LIN {X 0,Y 554.987,Z 579.027,A -85,B 0,C 180,E1 25629.323,E2 25629.323} C_VEL
LIN {X 0,Y 555.409,Z 560.565,A -85,B 0,C 180,E1 25628.677,E2 25628.677} C_VEL
LIN {X 0,Y 555.693,Z 541.746,A -85,B 0,C 180,E1 25628.23,E2 25628.23} C_VEL
LIN {X 0,Y 556.819,Z 343.095,A -85,B 0,C 180,E1 25625.485,E2 25625.485} C_VEL
LIN {X 0,Y 555.247,Z 334.788,A -85,B 0,C 180,E1 25625.25,E2 25625.25} C_VEL
LIN {X 0,Y 556.018,Z 305.385,A -85,B 0,C 180,E1 25622.475,E2 25622.475} C_VEL
LIN {X 0,Y 552.345,Z 293.887,A -85,B 0,C 180,E1 25621.069,E2 25621.069} C_VEL
LIN {X 0,Y 552.34,Z 293.681,A -85,B 0,C 180,E1 25617.846,E2 25617.846} C_VEL
LIN {X 0,Y 552.335,Z 293.677,A -85,B 0,C 180,E1 25614.474,E2 25614.474} C_VEL
LIN {X 0,Y 552.308,Z 293.678,A -85,B 0,C 180,E1 25611.119,E2 25611.119} C_VEL
LIN {X 0,Y 552.34,Z 293.682,A -85,B 0,C 180,E1 25607.811,E2 25607.811} C_VEL
LIN {X 0,Y 552.322,Z 293.677,A -85,B 0,C 180,E1 25604.474,E2 25604.474} C_VEL
LIN {X 0,Y 552.301,Z 293.684,A -85,B 0,C 180,E1 25601.084,E2 25601.084} C_VEL
LIN {X 0,Y 552.345,Z 293.682,A -85,B 0,C 180,E1 25597.855,E2 25597.855} C_VEL
LIN {X 0,Y 552.302,Z 293.681,A -85,B 0,C 180,E1 25594.545,E2 25594.545} C_VEL
LIN {X 0,Y 552.297,Z 293.685,A -85,B 0,C 180,E1 25591.099,E2 25591.099} C_VEL
LIN {X 0,Y 552.344,Z 293.681,A -85,B 0,C 180,E1 25587.842,E2 25587.842} C_VEL
LIN {X 0,Y 552.285,Z 293.679,A -85,B 0,C 180,E1 25584.607,E2 25584.607} C_VEL
LIN {X 0,Y 552.314,Z 293.685,A -85,B 0,C 180,E1 25581.338,E2 25581.338} C_VEL
LIN {X 0,Y 552.292,Z 293.682,A -85,B 0,C 180,E1 25578.252,E2 25578.252} C_VEL
LIN {X 0,Y 552.278,Z 293.681,A -85,B 0,C 180,E1 25574.897,E2 25574.897} C_VEL
LIN {X 0,Y 552.337,Z 293.685,A -85,B 0,C 180,E1 25571.676,E2 25571.676} C_VEL
LIN {X 0,Y 552.267,Z 293.68,A -85,B 0,C 180,E1 25568.433,E2 25568.433} C_VEL
LIN {X 0,Y 552.298,Z 293.687,A -85,B 0,C 180,E1 25565.194,E2 25565.194} C_VEL
LIN {X 0,Y 552.276,Z 293.682,A -85,B 0,C 180,E1 25562.075,E2 25562.075} C_VEL
LIN {X 0,Y 552.263,Z 293.686,A -85,B 0,C 180,E1 25558.755,E2 25558.755} C_VEL
LIN {X 0,Y 552.326,Z 293.685,A -85,B 0,C 180,E1 25555.536,E2 25555.536} C_VEL
LIN {X 0,Y 552.265,Z 293.683,A -85,B 0,C 180,E1 25552.406,E2 25552.406} C_VEL
LIN {X 0,Y 552.318,Z 293.686,A -85,B 0,C 180,E1 25549.148,E2 25549.148} C_VEL
LIN {X 0,Y 552.281,Z 293.681,A -85,B 0,C 180,E1 25546.014,E2 25546.014} C_VEL
LIN {X 0,Y 552.279,Z 293.683,A -85,B 0,C 180,E1 25542.566,E2 25542.566} C_VEL
LIN {X 0,Y 552.342,Z 293.686,A -85,B 0,C 180,E1 25539.33,E2 25539.33} C_VEL
LIN {X 0,Y 552.285,Z 293.683,A -85,B 0,C 180,E1 25536.096,E2 25536.096} C_VEL
LIN {X 0,Y 552.309,Z 293.68,A -85,B 0,C 180,E1 25532.741,E2 25532.741} C_VEL
LIN {X 0,Y 552.327,Z 293.686,A -85,B 0,C 180,E1 25529.504,E2 25529.504} C_VEL
LIN {X 0,Y 552.292,Z 293.684,A -85,B 0,C 180,E1 25526.195,E2 25526.195} C_VEL
LIN {X 0,Y 552.345,Z 293.677,A -85,B 0,C 180,E1 25522.93,E2 25522.93} C_VEL
LIN {X 0,Y 552.318,Z 293.684,A -85,B 0,C 180,E1 25519.603,E2 25519.603} C_VEL
LIN {X 0,Y 552.305,Z 293.684,A -85,B 0,C 180,E1 25516.245,E2 25516.245} C_VEL
LIN {X 0,Y 552.341,Z 293.676,A -85,B 0,C 180,E1 25513.002,E2 25513.002} C_VEL
LIN {X 0,Y 552.312,Z 293.674,A -85,B 0,C 180,E1 25509.702,E2 25509.702} C_VEL
LIN {X 0,Y 552.379,Z 293.923,A -85,B 0,C 180,E1 25506.704,E2 25506.704} C_VEL
LIN {X 0,Y 554.146,Z 298.811,A -85,B 0,C 180,E1 25506.242,E2 25506.242} C_VEL
LIN {X 0,Y 559.158,Z 310.667,A -85,B 0,C 180,E1 25505.196,E2 25505.196} C_VEL
LIN {X 0,Y 558.362,Z 353.988,A -85,B 0,C 180,E1 25502.614,E2 25502.614} C_VEL
LIN {X 0,Y 557.656,Z 390.963,A -85,B 0,C 180,E1 25500.436,E2 25500.436} C_VEL
LIN {X 0,Y 558.742,Z 400.337,A -85,B 0,C 180,E1 25500.232,E2 25500.232} C_VEL
LIN {X 0,Y 557.381,Z 635.152,A -85,B 0,C 180,E1 25496.937,E2 25496.937} C_VEL
LIN {X 0,Y 557.116,Z 659.61,A -85,B 0,C 180,E1 25496.529,E2 25496.529} C_VEL
LIN {X 0,Y 556.72,Z 680.633,A -85,B 0,C 180,E1 25495.975,E2 25495.975} C_VEL
LIN {X 0,Y 556.289,Z 700.028,A -85,B 0,C 180,E1 25495.274,E2 25495.274} C_VEL
LIN {X 0,Y 555.753,Z 719.239,A -85,B 0,C 180,E1 25494.386,E2 25494.386} C_VEL
LIN {X 0,Y 555.148,Z 738.316,A -85,B 0,C 180,E1 25493.286,E2 25493.286} C_VEL
LIN {X 0,Y 554.551,Z 756.388,A -85,B 0,C 180,E1 25492.025,E2 25492.025} C_VEL
LIN {X 0,Y 553.976,Z 773.443,A -85,B 0,C 180,E1 25490.606,E2 25490.606} C_VEL
LIN {X 0,Y 553.441,Z 789.448,A -85,B 0,C 180,E1 25489.031,E2 25489.031} C_VEL
LIN {X 0,Y 552.984,Z 804.238,A -85,B 0,C 180,E1 25487.315,E2 25487.315} C_VEL
LIN {X 0,Y 552.622,Z 817.278,A -85,B 0,C 180,E1 25485.531,E2 25485.531} C_VEL
LIN {X 0,Y 552.359,Z 828.534,A -85,B 0,C 180,E1 25483.717,E2 25483.717} C_VEL
LIN {X 0,Y 552.147,Z 838.91,A -85,B 0,C 180,E1 25481.701,E2 25481.701} C_VEL
LIN {X 0,Y 552.024,Z 847.28,A -85,B 0,C 180,E1 25479.697,E2 25479.697} C_VEL
LIN {X 0,Y 551.959,Z 854.202,A -85,B 0,C 180,E1 25477.599,E2 25477.599} C_VEL
LIN {X 0,Y 551.92,Z 859.556,A -85,B 0,C 180,E1 25475.405,E2 25475.405} C_VEL
LIN {X 0,Y 551.909,Z 862.942,A -85,B 0,C 180,E1 25473.323,E2 25473.323} C_VEL
LIN {X 0,Y 551.911,Z 864.759,A -85,B 0,C 180,E1 25471.142,E2 25471.142} C_VEL
LIN {X 0,Y 551.915,Z 864.783,A -85,B 0,C 180,E1 25468.962,E2 25468.962} C_VEL
LIN {X 0,Y 551.914,Z 863.169,A -85,B 0,C 180,E1 25466.885,E2 25466.885} C_VEL
LIN {X 0,Y 551.921,Z 859.76,A -85,B 0,C 180,E1 25464.699,E2 25464.699} C_VEL
LIN {X 0,Y 551.952,Z 854.809,A -85,B 0,C 180,E1 25462.611,E2 25462.611} C_VEL
LIN {X 0,Y 552.022,Z 848.49,A -85,B 0,C 180,E1 25460.618,E2 25460.618} C_VEL
LIN {X 0,Y 552.138,Z 839.875,A -85,B 0,C 180,E1 25458.51,E2 25458.51} C_VEL
LIN {X 0,Y 552.321,Z 830.266,A -85,B 0,C 180,E1 25456.602,E2 25456.602} C_VEL
LIN {X 0,Y 552.585,Z 818.607,A -85,B 0,C 180,E1 25454.67,E2 25454.67} C_VEL
LIN {X 0,Y 552.945,Z 805.602,A -85,B 0,C 180,E1 25452.858,E2 25452.858} C_VEL
LIN {X 0,Y 553.393,Z 790.965,A -85,B 0,C 180,E1 25451.131,E2 25451.131} C_VEL
LIN {X 0,Y 553.892,Z 775.855,A -85,B 0,C 180,E1 25449.611,E2 25449.611} C_VEL
LIN {X 0,Y 554.455,Z 759.284,A -85,B 0,C 180,E1 25448.193,E2 25448.193} C_VEL
LIN {X 0,Y 555.07,Z 740.902,A -85,B 0,C 180,E1 25446.879,E2 25446.879} C_VEL
LIN {X 0,Y 555.652,Z 722.284,A -85,B 0,C 180,E1 25445.779,E2 25445.779} C_VEL
LIN {X 0,Y 556.159,Z 704.004,A -85,B 0,C 180,E1 25444.896,E2 25444.896} C_VEL
LIN {X 0,Y 556.654,Z 683.569,A -85,B 0,C 180,E1 25444.118,E2 25444.118} C_VEL
LIN {X 0,Y 557.081,Z 663.506,A -85,B 0,C 180,E1 25443.556,E2 25443.556} C_VEL
LIN {X 0,Y 557.344,Z 642.37,A -85,B 0,C 180,E1 25443.163,E2 25443.163} C_VEL
LIN {X 0,Y 558.712,Z 404.697,A -85,B 0,C 180,E1 25439.829,E2 25439.829} C_VEL
LIN {X 0,Y 558.481,Z 396.637,A -85,B 0,C 180,E1 25439.698,E2 25439.698} C_VEL
LIN {X 0,Y 557.585,Z 389.593,A -85,B 0,C 180,E1 25439.505,E2 25439.505} C_VEL
LIN {X 0,Y 558.839,Z 332.018,A -85,B 0,C 180,E1 25436.068,E2 25436.068} C_VEL
LIN {X 0,Y 558.964,Z 309.864,A -85,B 0,C 180,E1 25434.743,E2 25434.743} C_VEL
LIN {X 0,Y 552.405,Z 294.092,A -85,B 0,C 180,E1 25433.324,E2 25433.324} C_VEL
LIN {X 0,Y 552.339,Z 293.671,A -85,B 0,C 180,E1 25432.969,E2 25432.969} C_VEL
LIN {X 0,Y 552.316,Z 293.676,A -85,B 0,C 180,E1 25429.653,E2 25429.653} C_VEL
LIN {X 0,Y 552.31,Z 293.676,A -85,B 0,C 180,E1 25426.246,E2 25426.246} C_VEL
LIN {X 0,Y 552.344,Z 293.682,A -85,B 0,C 180,E1 25423.004,E2 25423.004} C_VEL
LIN {X 0,Y 552.302,Z 293.683,A -85,B 0,C 180,E1 25419.702,E2 25419.702} C_VEL
LIN {X 0,Y 552.307,Z 293.672,A -85,B 0,C 180,E1 25416.297,E2 25416.297} C_VEL
LIN {X 0,Y 552.34,Z 293.682,A -85,B 0,C 180,E1 25413.016,E2 25413.016} C_VEL
LIN {X 0,Y 552.29,Z 293.685,A -85,B 0,C 180,E1 25409.739,E2 25409.739} C_VEL
LIN {X 0,Y 552.326,Z 293.687,A -85,B 0,C 180,E1 25406.444,E2 25406.444} C_VEL
LIN {X 0,Y 552.304,Z 293.681,A -85,B 0,C 180,E1 25403.244,E2 25403.244} C_VEL
LIN {X 0,Y 552.284,Z 293.685,A -85,B 0,C 180,E1 25399.898,E2 25399.898} C_VEL
LIN {X 0,Y 552.345,Z 293.684,A -85,B 0,C 180,E1 25396.619,E2 25396.619} C_VEL
LIN {X 0,Y 552.277,Z 293.679,A -85,B 0,C 180,E1 25393.399,E2 25393.399} C_VEL
LIN {X 0,Y 552.284,Z 293.685,A -85,B 0,C 180,E1 25389.992,E2 25389.992} C_VEL
LIN {X 0,Y 552.307,Z 293.682,A -85,B 0,C 180,E1 25386.862,E2 25386.862} C_VEL
LIN {X 0,Y 552.263,Z 293.684,A -85,B 0,C 180,E1 25383.633,E2 25383.633} C_VEL
LIN {X 0,Y 552.332,Z 293.688,A -85,B 0,C 180,E1 25380.415,E2 25380.415} C_VEL
LIN {X 0,Y 552.261,Z 293.683,A -85,B 0,C 180,E1 25377.198,E2 25377.198} C_VEL
LIN {X 0,Y 552.27,Z 293.687,A -85,B 0,C 180,E1 25373.764,E2 25373.764} C_VEL
LIN {X 0,Y 552.286,Z 293.681,A -85,B 0,C 180,E1 25370.833,E2 25370.833} C_VEL
LIN {X 0,Y 552.268,Z 293.686,A -85,B 0,C 180,E1 25367.558,E2 25367.558} C_VEL
LIN {X 0,Y 552.34,Z 293.683,A -85,B 0,C 180,E1 25364.352,E2 25364.352} C_VEL
LIN {X 0,Y 552.276,Z 293.684,A -85,B 0,C 180,E1 25361.091,E2 25361.091} C_VEL
LIN {X 0,Y 552.301,Z 293.685,A -85,B 0,C 180,E1 25357.767,E2 25357.767} C_VEL
LIN {X 0,Y 552.312,Z 293.681,A -85,B 0,C 180,E1 25354.593,E2 25354.593} C_VEL
LIN {X 0,Y 552.299,Z 293.687,A -85,B 0,C 180,E1 25352.738,E2 25352.738} C_VEL
LIN {X 0,Y 551.36,Z 293.809,A -85,B 0,C 180,E1 25351.938,E2 25351.938} C_VEL
LIN {X 0,Y 544.881,Z 294.609,A -85,B 0,C 180,E1 25349.694,E2 25349.694} C_VEL
LIN {X 0,Y 544.346,Z 294.673,A -85,B 0,C 180,E1 25349.109,E2 25349.109} C_VEL
LIN {X 0,Y 544.389,Z 294.67,A -85,B 0,C 180,E1 25345.804,E2 25345.804} C_VEL
LIN {X 0,Y 544.381,Z 294.675,A -85,B 0,C 180,E1 25342.507,E2 25342.507} C_VEL
LIN {X 0,Y 544.357,Z 294.672,A -85,B 0,C 180,E1 25339.164,E2 25339.164} C_VEL
LIN {X 0,Y 544.405,Z 294.667,A -85,B 0,C 180,E1 25335.887,E2 25335.887} C_VEL
LIN {X 0,Y 544.376,Z 294.665,A -85,B 0,C 180,E1 25332.523,E2 25332.523} C_VEL
LIN {X 0,Y 544.368,Z 294.665,A -85,B 0,C 180,E1 25329.184,E2 25329.184} C_VEL
LIN {X 0,Y 544.404,Z 294.669,A -85,B 0,C 180,E1 25325.864,E2 25325.864} C_VEL
LIN {X 0,Y 544.38,Z 294.676,A -85,B 0,C 180,E1 25322.537,E2 25322.537} C_VEL
LIN {X 0,Y 544.416,Z 294.861,A -85,B 0,C 180,E1 25319.297,E2 25319.297} C_VEL
LIN {X 0,Y 548.778,Z 308.855,A -85,B 0,C 180,E1 25317.566,E2 25317.566} C_VEL
LIN {X 0,Y 548.006,Z 335.919,A -85,B 0,C 180,E1 25315.02,E2 25315.02} C_VEL
LIN {X 0,Y 549.744,Z 345.387,A -85,B 0,C 180,E1 25314.785,E2 25314.785} C_VEL
LIN {X 0,Y 548.559,Z 542.987,A -85,B 0,C 180,E1 25312.041,E2 25312.041} C_VEL
LIN {X 0,Y 548.263,Z 561.882,A -85,B 0,C 180,E1 25311.584,E2 25311.584} C_VEL
LIN {X 0,Y 547.817,Z 579.557,A -85,B 0,C 180,E1 25310.96,E2 25310.96} C_VEL
LIN {X 0,Y 547.296,Z 596.827,A -85,B 0,C 180,E1 25310.146,E2 25310.146} C_VEL
LIN {X 0,Y 546.679,Z 613.249,A -85,B 0,C 180,E1 25309.165,E2 25309.165} C_VEL
LIN {X 0,Y 546.031,Z 629.329,A -85,B 0,C 180,E1 25307.971,E2 25307.971} C_VEL
LIN {X 0,Y 545.411,Z 644.251,A -85,B 0,C 180,E1 25306.617,E2 25306.617} C_VEL
LIN {X 0,Y 544.925,Z 659.491,A -85,B 0,C 180,E1 25304.993,E2 25304.993} C_VEL
LIN {X 0,Y 544.571,Z 672.136,A -85,B 0,C 180,E1 25303.376,E2 25303.376} C_VEL
LIN {X 0,Y 544.302,Z 683.234,A -85,B 0,C 180,E1 25301.657,E2 25301.657} C_VEL
LIN {X 0,Y 544.121,Z 692.806,A -85,B 0,C 180,E1 25299.84,E2 25299.84} C_VEL
LIN {X 0,Y 544.003,Z 700.413,A -85,B 0,C 180,E1 25298.029,E2 25298.029} C_VEL
LIN {X 0,Y 543.946,Z 706.59,A -85,B 0,C 180,E1 25296.12,E2 25296.12} C_VEL
LIN {X 0,Y 543.921,Z 710.996,A -85,B 0,C 180,E1 25294.217,E2 25294.217} C_VEL
LIN {X 0,Y 543.913,Z 713.744,A -85,B 0,C 180,E1 25292.318,E2 25292.318} C_VEL
LIN {X 0,Y 543.909,Z 714.928,A -85,B 0,C 180,E1 25290.316,E2 25290.316} C_VEL
LIN {X 0,Y 543.913,Z 714.376,A -85,B 0,C 180,E1 25288.315,E2 25288.315} C_VEL
LIN {X 0,Y 543.911,Z 712.229,A -85,B 0,C 180,E1 25286.417,E2 25286.417} C_VEL
LIN {X 0,Y 543.932,Z 708.459,A -85,B 0,C 180,E1 25284.515,E2 25284.515} C_VEL
LIN {X 0,Y 543.974,Z 702.972,A -85,B 0,C 180,E1 25282.608,E2 25282.608} C_VEL
LIN {X 0,Y 544.075,Z 695.621,A -85,B 0,C 180,E1 25280.694,E2 25280.694} C_VEL
LIN {X 0,Y 544.235,Z 686.506,A -85,B 0,C 180,E1 25278.831,E2 25278.831} C_VEL
LIN {X 0,Y 544.463,Z 676.445,A -85,B 0,C 180,E1 25277.162,E2 25277.162} C_VEL
LIN {X 0,Y 544.769,Z 664.701,A -85,B 0,C 180,E1 25275.546,E2 25275.546} C_VEL
LIN {X 0,Y 545.161,Z 651.496,A -85,B 0,C 180,E1 25274.032,E2 25274.032} C_VEL
LIN {X 0,Y 545.774,Z 635.715,A -85,B 0,C 180,E1 25272.484,E2 25272.484} C_VEL
LIN {X 0,Y 546.393,Z 620.716,A -85,B 0,C 180,E1 25271.268,E2 25271.268} C_VEL
LIN {X 0,Y 547.021,Z 604.25,A -85,B 0,C 180,E1 25270.181,E2 25270.181} C_VEL
LIN {X 0,Y 547.584,Z 587.755,A -85,B 0,C 180,E1 25269.31,E2 25269.31} C_VEL
LIN {X 0,Y 548.078,Z 569.85,A -85,B 0,C 180,E1 25268.584,E2 25268.584} C_VEL
LIN {X 0,Y 548.441,Z 551.518,A -85,B 0,C 180,E1 25268.051,E2 25268.051} C_VEL
LIN {X 0,Y 548.652,Z 532.068,A -85,B 0,C 180,E1 25267.695,E2 25267.695} C_VEL
LIN {X 0,Y 549.626,Z 343.643,A -85,B 0,C 180,E1 25265.094,E2 25265.094} C_VEL
LIN {X 0,Y 547.949,Z 335.49,A -85,B 0,C 180,E1 25264.869,E2 25264.869} C_VEL
LIN {X 0,Y 548.672,Z 308.058,A -85,B 0,C 180,E1 25262.257,E2 25262.257} C_VEL
LIN {X 0,Y 544.419,Z 294.84,A -85,B 0,C 180,E1 25260.606,E2 25260.606} C_VEL
LIN {X 0,Y 544.375,Z 294.675,A -85,B 0,C 180,E1 25257.193,E2 25257.193} C_VEL
LIN {X 0,Y 544.4,Z 294.672,A -85,B 0,C 180,E1 25253.876,E2 25253.876} C_VEL
LIN {X 0,Y 544.393,Z 294.662,A -85,B 0,C 180,E1 25250.48,E2 25250.48} C_VEL
LIN {X 0,Y 544.367,Z 294.663,A -85,B 0,C 180,E1 25247.127,E2 25247.127} C_VEL
LIN {X 0,Y 544.405,Z 294.671,A -85,B 0,C 180,E1 25243.8,E2 25243.8} C_VEL
LIN {X 0,Y 544.381,Z 294.669,A -85,B 0,C 180,E1 25240.418,E2 25240.418} C_VEL
LIN {X 0,Y 544.36,Z 294.674,A -85,B 0,C 180,E1 25237.046,E2 25237.046} C_VEL
LIN {X 0,Y 544.403,Z 294.67,A -85,B 0,C 180,E1 25233.699,E2 25233.699} C_VEL
LIN {X 0,Y 544.361,Z 294.671,A -85,B 0,C 180,E1 25230.461,E2 25230.461} C_VEL
LIN {X 0,Y 544.354,Z 294.675,A -85,B 0,C 180,E1 25227.025,E2 25227.025} C_VEL
LIN {X 0,Y 544.404,Z 294.668,A -85,B 0,C 180,E1 25223.717,E2 25223.717} C_VEL
LIN {X 0,Y 544.345,Z 294.671,A -85,B 0,C 180,E1 25220.488,E2 25220.488} C_VEL
LIN {X 0,Y 544.352,Z 294.676,A -85,B 0,C 180,E1 25217.091,E2 25217.091} C_VEL
LIN {X 0,Y 544.376,Z 294.667,A -85,B 0,C 180,E1 25213.923,E2 25213.923} C_VEL
LIN {X 0,Y 544.33,Z 294.675,A -85,B 0,C 180,E1 25210.676,E2 25210.676} C_VEL
LIN {X 0,Y 544.382,Z 294.675,A -85,B 0,C 180,E1 25207.387,E2 25207.387} C_VEL
LIN {X 0,Y 544.331,Z 294.675,A -85,B 0,C 180,E1 25204.214,E2 25204.214} C_VEL
LIN {X 0,Y 544.328,Z 294.677,A -85,B 0,C 180,E1 25200.842,E2 25200.842} C_VEL
LIN {X 0,Y 544.358,Z 294.674,A -85,B 0,C 180,E1 25197.79,E2 25197.79} C_VEL
LIN {X 0,Y 544.324,Z 294.676,A -85,B 0,C 180,E1 25194.519,E2 25194.519} C_VEL
LIN {X 0,Y 544.394,Z 294.67,A -85,B 0,C 180,E1 25191.338,E2 25191.338} C_VEL
LIN {X 0,Y 544.336,Z 294.676,A -85,B 0,C 180,E1 25188.128,E2 25188.128} C_VEL
LIN {X 0,Y 544.343,Z 294.675,A -85,B 0,C 180,E1 25184.644,E2 25184.644} C_VEL
LIN {X 0,Y 544.4,Z 294.669,A -85,B 0,C 180,E1 25181.382,E2 25181.382} C_VEL
LIN {X 0,Y 544.344,Z 294.675,A -85,B 0,C 180,E1 25178.107,E2 25178.107} C_VEL
LIN {X 0,Y 544.37,Z 294.673,A -85,B 0,C 180,E1 25174.779,E2 25174.779} C_VEL
LIN {X 0,Y 544.38,Z 294.673,A -85,B 0,C 180,E1 25171.595,E2 25171.595} C_VEL
LIN {X 0,Y 544.353,Z 294.672,A -85,B 0,C 180,E1 25168.256,E2 25168.256} C_VEL
LIN {X 0,Y 544.399,Z 294.657,A -85,B 0,C 180,E1 25164.91,E2 25164.91} C_VEL
LIN {X 0,Y 544.377,Z 294.673,A -85,B 0,C 180,E1 25161.625,E2 25161.625} C_VEL
LIN {X 0,Y 544.361,Z 294.657,A -85,B 0,C 180,E1 25158.219,E2 25158.219} C_VEL
LIN {X 0,Y 544.405,Z 294.666,A -85,B 0,C 180,E1 25154.997,E2 25154.997} C_VEL
LIN {X 0,Y 544.379,Z 294.677,A -85,B 0,C 180,E1 25151.623,E2 25151.623} C_VEL
LIN {X 0,Y 544.374,Z 294.678,A -85,B 0,C 180,E1 25148.177,E2 25148.177} C_VEL
LIN {X 0,Y 544.442,Z 294.964,A -85,B 0,C 180,E1 25147.17,E2 25147.17} C_VEL
LIN {X 0,Y 548.919,Z 306.372,A -85,B 0,C 180,E1 25146.115,E2 25146.115} C_VEL
LIN {X 0,Y 552.058,Z 313.827,A -85,B 0,C 180,E1 25145.452,E2 25145.452} C_VEL
LIN {X 0,Y 551.041,Z 367.835,A -85,B 0,C 180,E1 25142.238,E2 25142.238} C_VEL
LIN {X 0,Y 550.595,Z 391.148,A -85,B 0,C 180,E1 25140.865,E2 25140.865} C_VEL
LIN {X 0,Y 551.824,Z 401.323,A -85,B 0,C 180,E1 25140.637,E2 25140.637} C_VEL
LIN {X 0,Y 550.243,Z 636.347,A -85,B 0,C 180,E1 25137.298,E2 25137.298} C_VEL
LIN {X 0,Y 549.945,Z 659.772,A -85,B 0,C 180,E1 25136.898,E2 25136.898} C_VEL
LIN {X 0,Y 549.493,Z 680.847,A -85,B 0,C 180,E1 25136.336,E2 25136.336} C_VEL
LIN {X 0,Y 548.978,Z 700.613,A -85,B 0,C 180,E1 25135.609,E2 25135.609} C_VEL
LIN {X 0,Y 548.378,Z 719.24,A -85,B 0,C 180,E1 25134.736,E2 25134.736} C_VEL
LIN {X 0,Y 547.692,Z 738.326,A -85,B 0,C 180,E1 25133.622,E2 25133.622} C_VEL
LIN {X 0,Y 546.999,Z 756.39,A -85,B 0,C 180,E1 25132.346,E2 25132.346} C_VEL
LIN {X 0,Y 546.323,Z 773.443,A -85,B 0,C 180,E1 25130.908,E2 25130.908} C_VEL
LIN {X 0,Y 545.715,Z 789.202,A -85,B 0,C 180,E1 25129.338,E2 25129.338} C_VEL
LIN {X 0,Y 545.179,Z 803.91,A -85,B 0,C 180,E1 25127.614,E2 25127.614} C_VEL
LIN {X 0,Y 544.775,Z 816.573,A -85,B 0,C 180,E1 25125.87,E2 25125.87} C_VEL
LIN {X 0,Y 544.438,Z 828.535,A -85,B 0,C 180,E1 25123.92,E2 25123.92} C_VEL
LIN {X 0,Y 544.188,Z 838.909,A -85,B 0,C 180,E1 25121.875,E2 25121.875} C_VEL
LIN {X 0,Y 544.043,Z 847.279,A -85,B 0,C 180,E1 25119.841,E2 25119.841} C_VEL
LIN {X 0,Y 543.968,Z 854.202,A -85,B 0,C 180,E1 25117.711,E2 25117.711} C_VEL
LIN {X 0,Y 543.923,Z 859.556,A -85,B 0,C 180,E1 25115.485,E2 25115.485} C_VEL
LIN {X 0,Y 543.909,Z 862.942,A -85,B 0,C 180,E1 25113.372,E2 25113.372} C_VEL
LIN {X 0,Y 543.91,Z 864.759,A -85,B 0,C 180,E1 25111.159,E2 25111.159} C_VEL
LIN {X 0,Y 543.914,Z 864.783,A -85,B 0,C 180,E1 25108.947,E2 25108.947} C_VEL
LIN {X 0,Y 543.913,Z 863.168,A -85,B 0,C 180,E1 25106.839,E2 25106.839} C_VEL
LIN {X 0,Y 543.922,Z 859.761,A -85,B 0,C 180,E1 25104.621,E2 25104.621} C_VEL
LIN {X 0,Y 543.96,Z 854.81,A -85,B 0,C 180,E1 25102.501,E2 25102.501} C_VEL
LIN {X 0,Y 544.038,Z 848.49,A -85,B 0,C 180,E1 25100.479,E2 25100.479} C_VEL
LIN {X 0,Y 544.175,Z 839.876,A -85,B 0,C 180,E1 25098.34,E2 25098.34} C_VEL
LIN {X 0,Y 544.394,Z 830.268,A -85,B 0,C 180,E1 25096.403,E2 25096.403} C_VEL
LIN {X 0,Y 544.705,Z 818.691,A -85,B 0,C 180,E1 25094.455,E2 25094.455} C_VEL
LIN {X 0,Y 545.128,Z 805.601,A -85,B 0,C 180,E1 25092.605,E2 25092.605} C_VEL
LIN {X 0,Y 545.651,Z 790.965,A -85,B 0,C 180,E1 25090.853,E2 25090.853} C_VEL
LIN {X 0,Y 546.252,Z 775.515,A -85,B 0,C 180,E1 25089.282,E2 25089.282} C_VEL
LIN {X 0,Y 546.907,Z 758.842,A -85,B 0,C 180,E1 25087.841,E2 25087.841} C_VEL
LIN {X 0,Y 547.591,Z 740.898,A -85,B 0,C 180,E1 25086.544,E2 25086.544} C_VEL
LIN {X 0,Y 548.224,Z 723.385,A -85,B 0,C 180,E1 25085.492,E2 25085.492} C_VEL
LIN {X 0,Y 548.857,Z 704.001,A -85,B 0,C 180,E1 25084.538,E2 25084.538} C_VEL
LIN {X 0,Y 549.412,Z 683.823,A -85,B 0,C 180,E1 25083.76,E2 25083.76} C_VEL
LIN {X 0,Y 549.903,Z 663.669,A -85,B 0,C 180,E1 25083.187,E2 25083.187} C_VEL
LIN {X 0,Y 550.205,Z 642.495,A -85,B 0,C 180,E1 25082.788,E2 25082.788} C_VEL
LIN {X 0,Y 551.793,Z 405.141,A -85,B 0,C 180,E1 25079.417,E2 25079.417} C_VEL
LIN {X 0,Y 551.569,Z 397.823,A -85,B 0,C 180,E1 25079.295,E2 25079.295} C_VEL
LIN {X 0,Y 550.502,Z 389.593,A -85,B 0,C 180,E1 25079.07,E2 25079.07} C_VEL
LIN {X 0,Y 551.484,Z 344.188,A -85,B 0,C 180,E1 25076.367,E2 25076.367} C_VEL
LIN {X 0,Y 551.986,Z 313.279,A -85,B 0,C 180,E1 25074.51,E2 25074.51} C_VEL
LIN {X 0,Y 544.464,Z 295.085,A -85,B 0,C 180,E1 25072.844,E2 25072.844} C_VEL
LIN {X 0,Y 544.387,Z 294.664,A -85,B 0,C 180,E1 25072.508,E2 25072.508} C_VEL
LIN {X 0,Y 544.405,Z 294.663,A -85,B 0,C 180,E1 25069.17,E2 25069.17} C_VEL
LIN {X 0,Y 544.365,Z 294.666,A -85,B 0,C 180,E1 25065.885,E2 25065.885} C_VEL
LIN {X 0,Y 544.388,Z 294.66,A -85,B 0,C 180,E1 25062.523,E2 25062.523} C_VEL
LIN {X 0,Y 544.401,Z 294.67,A -85,B 0,C 180,E1 25059.183,E2 25059.183} C_VEL
LIN {X 0,Y 544.354,Z 294.66,A -85,B 0,C 180,E1 25055.869,E2 25055.869} C_VEL
LIN {X 0,Y 544.393,Z 294.676,A -85,B 0,C 180,E1 25052.542,E2 25052.542} C_VEL
LIN {X 0,Y 544.376,Z 294.672,A -85,B 0,C 180,E1 25049.246,E2 25049.246} C_VEL
LIN {X 0,Y 544.349,Z 294.675,A -85,B 0,C 180,E1 25045.922,E2 25045.922} C_VEL
LIN {X 0,Y 544.409,Z 294.668,A -85,B 0,C 180,E1 25042.686,E2 25042.686} C_VEL
LIN {X 0,Y 544.348,Z 294.672,A -85,B 0,C 180,E1 25039.418,E2 25039.418} C_VEL
LIN {X 0,Y 544.349,Z 294.676,A -85,B 0,C 180,E1 25035.993,E2 25035.993} C_VEL
LIN {X 0,Y 544.397,Z 294.666,A -85,B 0,C 180,E1 25032.732,E2 25032.732} C_VEL
LIN {X 0,Y 544.333,Z 294.673,A -85,B 0,C 180,E1 25029.474,E2 25029.474} C_VEL
LIN {X 0,Y 544.366,Z 294.677,A -85,B 0,C 180,E1 25026.221,E2 25026.221} C_VEL
LIN {X 0,Y 544.342,Z 294.672,A -85,B 0,C 180,E1 25023.053,E2 25023.053} C_VEL
LIN {X 0,Y 544.324,Z 294.677,A -85,B 0,C 180,E1 25019.684,E2 25019.684} C_VEL
LIN {X 0,Y 544.383,Z 294.669,A -85,B 0,C 180,E1 25016.525,E2 25016.525} C_VEL
LIN {X 0,Y 544.321,Z 294.676,A -85,B 0,C 180,E1 25013.354,E2 25013.354} C_VEL
LIN {X 0,Y 544.376,Z 294.675,A -85,B 0,C 180,E1 25010.165,E2 25010.165} C_VEL
LIN {X 0,Y 544.335,Z 294.675,A -85,B 0,C 180,E1 25007.05,E2 25007.05} C_VEL
LIN {X 0,Y 544.338,Z 294.675,A -85,B 0,C 180,E1 25003.568,E2 25003.568} C_VEL
LIN {X 0,Y 544.397,Z 294.669,A -85,B 0,C 180,E1 25000.36,E2 25000.36} C_VEL
LIN {X 0,Y 544.34,Z 294.675,A -85,B 0,C 180,E1 24997.082,E2 24997.082} C_VEL
LIN {X 0,Y 544.361,Z 294.673,A -85,B 0,C 180,E1 24993.677,E2 24993.677} C_VEL
LIN {X 0,Y 544.38,Z 294.672,A -85,B 0,C 180,E1 24990.512,E2 24990.512} C_VEL
LIN {X 0,Y 544.346,Z 294.673,A -85,B 0,C 180,E1 24989.109,E2 24989.109} C_VEL
LIN {X 0,Y 543.375,Z 294.804,A -85,B 0,C 180,E1 24988.298,E2 24988.298} C_VEL
LIN {X 0,Y 536.878,Z 295.607,A -85,B 0,C 180,E1 24985.962,E2 24985.962} C_VEL
LIN {X 0,Y 536.42,Z 295.66,A -85,B 0,C 180,E1 24985.427,E2 24985.427} C_VEL
LIN {X 0,Y 536.466,Z 295.659,A -85,B 0,C 180,E1 24982.179,E2 24982.179} C_VEL
LIN {X 0,Y 536.421,Z 295.663,A -85,B 0,C 180,E1 24978.852,E2 24978.852} C_VEL
LIN {X 0,Y 536.433,Z 295.656,A -85,B 0,C 180,E1 24975.397,E2 24975.397} C_VEL
LIN {X 0,Y 536.464,Z 295.657,A -85,B 0,C 180,E1 24972.116,E2 24972.116} C_VEL
LIN {X 0,Y 536.426,Z 295.652,A -85,B 0,C 180,E1 24968.775,E2 24968.775} C_VEL
LIN {X 0,Y 536.442,Z 295.657,A -85,B 0,C 180,E1 24965.295,E2 24965.295} C_VEL
LIN {X 0,Y 536.463,Z 295.656,A -85,B 0,C 180,E1 24961.958,E2 24961.958} C_VEL
LIN {X 0,Y 536.499,Z 295.915,A -85,B 0,C 180,E1 24959.745,E2 24959.745} C_VEL
LIN {X 0,Y 541.485,Z 311.262,A -85,B 0,C 180,E1 24957.812,E2 24957.812} C_VEL
LIN {X 0,Y 540.72,Z 336.313,A -85,B 0,C 180,E1 24955.435,E2 24955.435} C_VEL
LIN {X 0,Y 542.697,Z 346.672,A -85,B 0,C 180,E1 24955.169,E2 24955.169} C_VEL
LIN {X 0,Y 541.466,Z 544.211,A -85,B 0,C 180,E1 24952.415,E2 24952.415} C_VEL
LIN {X 0,Y 541.155,Z 563.162,A -85,B 0,C 180,E1 24951.949,E2 24951.949} C_VEL
LIN {X 0,Y 540.667,Z 580.996,A -85,B 0,C 180,E1 24951.308,E2 24951.308} C_VEL
LIN {X 0,Y 540.083,Z 598.216,A -85,B 0,C 180,E1 24950.48,E2 24950.48} C_VEL
LIN {X 0,Y 539.356,Z 615.276,A -85,B 0,C 180,E1 24949.436,E2 24949.436} C_VEL
LIN {X 0,Y 538.667,Z 630.549,A -85,B 0,C 180,E1 24948.281,E2 24948.281} C_VEL
LIN {X 0,Y 537.958,Z 645.447,A -85,B 0,C 180,E1 24946.91,E2 24946.91} C_VEL
LIN {X 0,Y 537.315,Z 658.759,A -85,B 0,C 180,E1 24945.432,E2 24945.432} C_VEL
LIN {X 0,Y 536.769,Z 671.005,A -85,B 0,C 180,E1 24943.794,E2 24943.794} C_VEL
LIN {X 0,Y 536.337,Z 684.507,A -85,B 0,C 180,E1 24941.615,E2 24941.615} C_VEL
LIN {X 0,Y 536.133,Z 693.838,A -85,B 0,C 180,E1 24939.771,E2 24939.771} C_VEL
LIN {X 0,Y 536.006,Z 701.614,A -85,B 0,C 180,E1 24937.826,E2 24937.826} C_VEL
LIN {X 0,Y 535.94,Z 707.481,A -85,B 0,C 180,E1 24935.889,E2 24935.889} C_VEL
LIN {X 0,Y 535.92,Z 711.772,A -85,B 0,C 180,E1 24933.851,E2 24933.851} C_VEL
LIN {X 0,Y 535.913,Z 714.248,A -85,B 0,C 180,E1 24931.818,E2 24931.818} C_VEL
LIN {X 0,Y 535.913,Z 714.969,A -85,B 0,C 180,E1 24929.786,E2 24929.786} C_VEL
LIN {X 0,Y 535.916,Z 713.954,A -85,B 0,C 180,E1 24927.755,E2 24927.755} C_VEL
LIN {X 0,Y 535.922,Z 711.375,A -85,B 0,C 180,E1 24925.828,E2 24925.828} C_VEL
LIN {X 0,Y 535.947,Z 707.148,A -85,B 0,C 180,E1 24923.896,E2 24923.896} C_VEL
LIN {X 0,Y 536.013,Z 701.161,A -85,B 0,C 180,E1 24921.958,E2 24921.958} C_VEL
LIN {X 0,Y 536.136,Z 693.754,A -85,B 0,C 180,E1 24920.121,E2 24920.121} C_VEL
LIN {X 0,Y 536.341,Z 684.398,A -85,B 0,C 180,E1 24918.276,E2 24918.276} C_VEL
LIN {X 0,Y 536.794,Z 670.46,A -85,B 0,C 180,E1 24916.035,E2 24916.035} C_VEL
LIN {X 0,Y 537.325,Z 658.594,A -85,B 0,C 180,E1 24914.458,E2 24914.458} C_VEL
LIN {X 0,Y 537.971,Z 645.245,A -85,B 0,C 180,E1 24912.979,E2 24912.979} C_VEL
LIN {X 0,Y 538.681,Z 630.3,A -85,B 0,C 180,E1 24911.607,E2 24911.607} C_VEL
LIN {X 0,Y 539.414,Z 614.175,A -85,B 0,C 180,E1 24910.398,E2 24910.398} C_VEL
LIN {X 0,Y 540.101,Z 597.813,A -85,B 0,C 180,E1 24909.407,E2 24909.407} C_VEL
LIN {X 0,Y 540.692,Z 580.44,A -85,B 0,C 180,E1 24908.579,E2 24908.579} C_VEL
LIN {X 0,Y 541.172,Z 562.076,A -85,B 0,C 180,E1 24907.93,E2 24907.93} C_VEL
LIN {X 0,Y 541.473,Z 543.525,A -85,B 0,C 180,E1 24907.484,E2 24907.484} C_VEL
LIN {X 0,Y 542.586,Z 364.02,A -85,B 0,C 180,E1 24904.978,E2 24904.978} C_VEL
LIN {X 0,Y 542.483,Z 344.395,A -85,B 0,C 180,E1 24904.696,E2 24904.696} C_VEL
LIN {X 0,Y 540.658,Z 335.774,A -85,B 0,C 180,E1 24904.445,E2 24904.445} C_VEL
LIN {X 0,Y 541.472,Z 311.202,A -85,B 0,C 180,E1 24902.09,E2 24902.09} C_VEL
LIN {X 0,Y 536.494,Z 295.899,A -85,B 0,C 180,E1 24900.159,E2 24900.159} C_VEL
LIN {X 0,Y 536.439,Z 295.662,A -85,B 0,C 180,E1 24896.9,E2 24896.9} C_VEL
LIN {X 0,Y 536.442,Z 295.663,A -85,B 0,C 180,E1 24893.386,E2 24893.386} C_VEL
LIN {X 0,Y 536.462,Z 295.654,A -85,B 0,C 180,E1 24889.985,E2 24889.985} C_VEL
LIN {X 0,Y 536.436,Z 295.648,A -85,B 0,C 180,E1 24886.629,E2 24886.629} C_VEL
LIN {X 0,Y 536.428,Z 295.664,A -85,B 0,C 180,E1 24883.162,E2 24883.162} C_VEL
LIN {X 0,Y 536.467,Z 295.661,A -85,B 0,C 180,E1 24879.838,E2 24879.838} C_VEL
LIN {X 0,Y 536.431,Z 295.66,A -85,B 0,C 180,E1 24876.484,E2 24876.484} C_VEL
LIN {X 0,Y 536.42,Z 295.663,A -85,B 0,C 180,E1 24873.103,E2 24873.103} C_VEL
LIN {X 0,Y 536.469,Z 295.658,A -85,B 0,C 180,E1 24869.844,E2 24869.844} C_VEL
LIN {X 0,Y 536.413,Z 295.662,A -85,B 0,C 180,E1 24866.533,E2 24866.533} C_VEL
LIN {X 0,Y 536.414,Z 295.664,A -85,B 0,C 180,E1 24863.044,E2 24863.044} C_VEL
LIN {X 0,Y 536.466,Z 295.656,A -85,B 0,C 180,E1 24859.749,E2 24859.749} C_VEL
LIN {X 0,Y 536.401,Z 295.663,A -85,B 0,C 180,E1 24856.459,E2 24856.459} C_VEL
LIN {X 0,Y 536.407,Z 295.664,A -85,B 0,C 180,E1 24853.035,E2 24853.035} C_VEL
LIN {X 0,Y 536.433,Z 295.663,A -85,B 0,C 180,E1 24849.874,E2 24849.874} C_VEL
LIN {X 0,Y 536.387,Z 295.665,A -85,B 0,C 180,E1 24846.637,E2 24846.637} C_VEL
LIN {X 0,Y 536.443,Z 295.657,A -85,B 0,C 180,E1 24843.42,E2 24843.42} C_VEL
LIN {X 0,Y 536.385,Z 295.666,A -85,B 0,C 180,E1 24840.214,E2 24840.214} C_VEL
LIN {X 0,Y 536.39,Z 295.661,A -85,B 0,C 180,E1 24836.794,E2 24836.794} C_VEL
LIN {X 0,Y 536.446,Z 295.665,A -85,B 0,C 180,E1 24833.579,E2 24833.579} C_VEL
LIN {X 0,Y 536.39,Z 295.663,A -85,B 0,C 180,E1 24830.342,E2 24830.342} C_VEL
LIN {X 0,Y 536.435,Z 295.655,A -85,B 0,C 180,E1 24827.076,E2 24827.076} C_VEL
LIN {X 0,Y 536.414,Z 295.665,A -85,B 0,C 180,E1 24823.875,E2 24823.875} C_VEL
LIN {X 0,Y 536.405,Z 295.662,A -85,B 0,C 180,E1 24820.509,E2 24820.509} C_VEL
LIN {X 0,Y 536.467,Z 295.656,A -85,B 0,C 180,E1 24817.191,E2 24817.191} C_VEL
LIN {X 0,Y 536.417,Z 295.664,A -85,B 0,C 180,E1 24813.903,E2 24813.903} C_VEL
LIN {X 0,Y 536.42,Z 295.662,A -85,B 0,C 180,E1 24810.509,E2 24810.509} C_VEL
LIN {X 0,Y 536.468,Z 295.662,A -85,B 0,C 180,E1 24807.197,E2 24807.197} C_VEL
LIN {X 0,Y 536.419,Z 295.646,A -85,B 0,C 180,E1 24803.914,E2 24803.914} C_VEL
LIN {X 0,Y 536.434,Z 295.66,A -85,B 0,C 180,E1 24800.501,E2 24800.501} C_VEL
LIN {X 0,Y 536.463,Z 295.652,A -85,B 0,C 180,E1 24797.134,E2 24797.134} C_VEL
LIN {X 0,Y 536.432,Z 295.65,A -85,B 0,C 180,E1 24793.748,E2 24793.748} C_VEL
LIN {X 0,Y 536.436,Z 295.65,A -85,B 0,C 180,E1 24790.297,E2 24790.297} C_VEL
LIN {X 0,Y 536.468,Z 295.89,A -85,B 0,C 180,E1 24787.684,E2 24787.684} C_VEL
LIN {X 0,Y 537.386,Z 298.529,A -85,B 0,C 180,E1 24787.395,E2 24787.395} C_VEL
LIN {X 0,Y 544.954,Z 316.732,A -85,B 0,C 180,E1 24785.725,E2 24785.725} C_VEL
LIN {X 0,Y 543.784,Z 370.83,A -85,B 0,C 180,E1 24782.472,E2 24782.472} C_VEL
LIN {X 0,Y 543.515,Z 391.139,A -85,B 0,C 180,E1 24781.306,E2 24781.306} C_VEL
LIN {X 0,Y 544.931,Z 402.537,A -85,B 0,C 180,E1 24781.049,E2 24781.049} C_VEL
LIN {X 0,Y 543.124,Z 637.969,A -85,B 0,C 180,E1 24777.663,E2 24777.663} C_VEL
LIN {X 0,Y 542.789,Z 660.42,A -85,B 0,C 180,E1 24777.267,E2 24777.267} C_VEL
LIN {X 0,Y 542.279,Z 681.388,A -85,B 0,C 180,E1 24776.695,E2 24776.695} C_VEL
LIN {X 0,Y 541.676,Z 701.436,A -85,B 0,C 180,E1 24775.942,E2 24775.942} C_VEL
LIN {X 0,Y 540.985,Z 720.276,A -85,B 0,C 180,E1 24775.039,E2 24775.039} C_VEL
LIN {X 0,Y 540.22,Z 739.219,A -85,B 0,C 180,E1 24773.911,E2 24773.911} C_VEL
LIN {X 0,Y 539.435,Z 757.064,A -85,B 0,C 180,E1 24772.623,E2 24772.623} C_VEL
LIN {X 0,Y 538.666,Z 774.049,A -85,B 0,C 180,E1 24771.163,E2 24771.163} C_VEL
LIN {X 0,Y 537.963,Z 789.953,A -85,B 0,C 180,E1 24769.544,E2 24769.544} C_VEL
LIN {X 0,Y 537.346,Z 804.756,A -85,B 0,C 180,E1 24767.767,E2 24767.767} C_VEL
LIN {X 0,Y 536.86,Z 817.987,A -85,B 0,C 180,E1 24765.889,E2 24765.889} C_VEL
LIN {X 0,Y 536.505,Z 829.114,A -85,B 0,C 180,E1 24764.02,E2 24764.02} C_VEL
LIN {X 0,Y 536.225,Z 839.412,A -85,B 0,C 180,E1 24761.945,E2 24761.945} C_VEL
LIN {X 0,Y 536.056,Z 848.088,A -85,B 0,C 180,E1 24759.772,E2 24759.772} C_VEL
LIN {X 0,Y 535.974,Z 854.505,A -85,B 0,C 180,E1 24757.719,E2 24757.719} C_VEL
LIN {X 0,Y 535.928,Z 859.555,A -85,B 0,C 180,E1 24755.567,E2 24755.567} C_VEL
LIN {X 0,Y 535.91,Z 862.941,A -85,B 0,C 180,E1 24753.423,E2 24753.423} C_VEL
LIN {X 0,Y 535.909,Z 864.759,A -85,B 0,C 180,E1 24751.176,E2 24751.176} C_VEL
LIN {X 0,Y 535.915,Z 864.805,A -85,B 0,C 180,E1 24749.038,E2 24749.038} C_VEL
LIN {X 0,Y 535.914,Z 863.281,A -85,B 0,C 180,E1 24746.899,E2 24746.899} C_VEL
LIN {X 0,Y 535.924,Z 859.966,A -85,B 0,C 180,E1 24744.648,E2 24744.648} C_VEL
LIN {X 0,Y 535.965,Z 855.113,A -85,B 0,C 180,E1 24742.497,E2 24742.497} C_VEL
LIN {X 0,Y 536.055,Z 848.49,A -85,B 0,C 180,E1 24740.336,E2 24740.336} C_VEL
LIN {X 0,Y 536.214,Z 839.877,A -85,B 0,C 180,E1 24738.164,E2 24738.164} C_VEL
LIN {X 0,Y 536.475,Z 830.125,A -85,B 0,C 180,E1 24736.171,E2 24736.171} C_VEL
LIN {X 0,Y 536.835,Z 818.69,A -85,B 0,C 180,E1 24734.222,E2 24734.222} C_VEL
LIN {X 0,Y 537.324,Z 805.371,A -85,B 0,C 180,E1 24732.313,E2 24732.313} C_VEL
LIN {X 0,Y 537.923,Z 790.965,A -85,B 0,C 180,E1 24730.567,E2 24730.567} C_VEL
LIN {X 0,Y 538.596,Z 775.859,A -85,B 0,C 180,E1 24729.006,E2 24729.006} C_VEL
LIN {X 0,Y 539.375,Z 758.573,A -85,B 0,C 180,E1 24727.494,E2 24727.494} C_VEL
LIN {X 0,Y 540.137,Z 740.895,A -85,B 0,C 180,E1 24726.201,E2 24726.201} C_VEL
LIN {X 0,Y 540.87,Z 722.982,A -85,B 0,C 180,E1 24725.114,E2 24725.114} C_VEL
LIN {X 0,Y 541.577,Z 703.998,A -85,B 0,C 180,E1 24724.171,E2 24724.171} C_VEL
LIN {X 0,Y 542.2,Z 683.938,A -85,B 0,C 180,E1 24723.387,E2 24723.387} C_VEL
LIN {X 0,Y 542.749,Z 663.832,A -85,B 0,C 180,E1 24722.808,E2 24722.808} C_VEL
LIN {X 0,Y 543.092,Z 642.495,A -85,B 0,C 180,E1 24722.402,E2 24722.402} C_VEL
LIN {X 0,Y 544.906,Z 405.395,A -85,B 0,C 180,E1 24718.992,E2 24718.992} C_VEL
LIN {X 0,Y 544.666,Z 398.89,A -85,B 0,C 180,E1 24718.879,E2 24718.879} C_VEL
LIN {X 0,Y 543.416,Z 389.969,A -85,B 0,C 180,E1 24718.652,E2 24718.652} C_VEL
LIN {X 0,Y 544.565,Z 334.264,A -85,B 0,C 180,E1 24715.341,E2 24715.341} C_VEL
LIN {X 0,Y 544.752,Z 316.051,A -85,B 0,C 180,E1 24714.219,E2 24714.219} C_VEL
LIN {X 0,Y 536.504,Z 296.088,A -85,B 0,C 180,E1 24712.353,E2 24712.353} C_VEL
LIN {X 0,Y 536.431,Z 295.662,A -85,B 0,C 180,E1 24712.039,E2 24712.039} C_VEL
LIN {X 0,Y 536.464,Z 295.66,A -85,B 0,C 180,E1 24708.686,E2 24708.686} C_VEL
LIN {X 0,Y 536.462,Z 295.652,A -85,B 0,C 180,E1 24705.211,E2 24705.211} C_VEL
LIN {X 0,Y 536.422,Z 295.643,A -85,B 0,C 180,E1 24701.858,E2 24701.858} C_VEL
LIN {X 0,Y 536.448,Z 295.662,A -85,B 0,C 180,E1 24698.483,E2 24698.483} C_VEL
LIN {X 0,Y 536.458,Z 295.644,A -85,B 0,C 180,E1 24695.096,E2 24695.096} C_VEL
LIN {X 0,Y 536.415,Z 295.661,A -85,B 0,C 180,E1 24691.795,E2 24691.795} C_VEL
LIN {X 0,Y 536.455,Z 295.662,A -85,B 0,C 180,E1 24688.499,E2 24688.499} C_VEL
LIN {X 0,Y 536.439,Z 295.662,A -85,B 0,C 180,E1 24685.148,E2 24685.148} C_VEL
LIN {X 0,Y 536.407,Z 295.664,A -85,B 0,C 180,E1 24681.838,E2 24681.838} C_VEL
LIN {X 0,Y 536.461,Z 295.657,A -85,B 0,C 180,E1 24678.585,E2 24678.585} C_VEL
LIN {X 0,Y 536.406,Z 295.663,A -85,B 0,C 180,E1 24675.348,E2 24675.348} C_VEL
LIN {X 0,Y 536.4,Z 295.665,A -85,B 0,C 180,E1 24671.88,E2 24671.88} C_VEL
LIN {X 0,Y 536.459,Z 295.657,A -85,B 0,C 180,E1 24668.575,E2 24668.575} C_VEL
LIN {X 0,Y 536.391,Z 295.665,A -85,B 0,C 180,E1 24665.348,E2 24665.348} C_VEL
LIN {X 0,Y 536.4,Z 295.663,A -85,B 0,C 180,E1 24661.923,E2 24661.923} C_VEL
LIN {X 0,Y 536.415,Z 295.666,A -85,B 0,C 180,E1 24658.825,E2 24658.825} C_VEL
LIN {X 0,Y 536.38,Z 295.665,A -85,B 0,C 180,E1 24655.509,E2 24655.509} C_VEL
LIN {X 0,Y 536.449,Z 295.656,A -85,B 0,C 180,E1 24652.288,E2 24652.288} C_VEL
LIN {X 0,Y 536.396,Z 295.665,A -85,B 0,C 180,E1 24649.039,E2 24649.039} C_VEL
LIN {X 0,Y 536.399,Z 295.657,A -85,B 0,C 180,E1 24645.646,E2 24645.646} C_VEL
LIN {X 0,Y 536.453,Z 295.665,A -85,B 0,C 180,E1 24642.426,E2 24642.426} C_VEL
LIN {X 0,Y 536.399,Z 295.661,A -85,B 0,C 180,E1 24639.143,E2 24639.143} C_VEL
LIN {X 0,Y 536.427,Z 295.655,A -85,B 0,C 180,E1 24635.791,E2 24635.791} C_VEL
LIN {X 0,Y 536.442,Z 295.665,A -85,B 0,C 180,E1 24632.521,E2 24632.521} C_VEL
LIN {X 0,Y 536.408,Z 295.662,A -85,B 0,C 180,E1 24629.235,E2 24629.235} C_VEL
LIN {X 0,Y 536.462,Z 295.658,A -85,B 0,C 180,E1 24626.003,E2 24626.003} C_VEL
LIN {X 0,Y 536.42,Z 295.66,A -85,B 0,C 180,E1 24625.427,E2 24625.427} C_VEL
LIN {X 0,Y 535.423,Z 295.79,A -85,B 0,C 180,E1 24624.605,E2 24624.605} C_VEL
LIN {X 0,Y 528.977,Z 296.593,A -85,B 0,C 180,E1 24622.234,E2 24622.234} C_VEL
LIN {X 0,Y 528.507,Z 296.648,A -85,B 0,C 180,E1 24621.691,E2 24621.691} C_VEL
LIN {X 0,Y 528.517,Z 296.649,A -85,B 0,C 180,E1 24618.353,E2 24618.353} C_VEL
LIN {X 0,Y 528.483,Z 296.646,A -85,B 0,C 180,E1 24614.961,E2 24614.961} C_VEL
LIN {X 0,Y 528.518,Z 296.65,A -85,B 0,C 180,E1 24611.606,E2 24611.606} C_VEL
LIN {X 0,Y 528.523,Z 296.635,A -85,B 0,C 180,E1 24608.214,E2 24608.214} C_VEL
LIN {X 0,Y 528.49,Z 296.642,A -85,B 0,C 180,E1 24604.805,E2 24604.805} C_VEL
LIN {X 0,Y 528.511,Z 296.637,A -85,B 0,C 180,E1 24601.348,E2 24601.348} C_VEL
LIN {X 0,Y 528.551,Z 296.858,A -85,B 0,C 180,E1 24600.242,E2 24600.242} C_VEL
LIN {X 0,Y 534.193,Z 314.111,A -85,B 0,C 180,E1 24598.021,E2 24598.021} C_VEL
LIN {X 0,Y 533.42,Z 336.395,A -85,B 0,C 180,E1 24595.877,E2 24595.877} C_VEL
LIN {X 0,Y 535.67,Z 347.817,A -85,B 0,C 180,E1 24595.564,E2 24595.564} C_VEL
LIN {X 0,Y 534.4,Z 545.275,A -85,B 0,C 180,E1 24592.802,E2 24592.802} C_VEL
LIN {X 0,Y 534.083,Z 564.213,A -85,B 0,C 180,E1 24592.332,E2 24592.332} C_VEL
LIN {X 0,Y 533.546,Z 582.504,A -85,B 0,C 180,E1 24591.664,E2 24591.664} C_VEL
LIN {X 0,Y 532.91,Z 599.652,A -85,B 0,C 180,E1 24590.826,E2 24590.826} C_VEL
LIN {X 0,Y 532.155,Z 615.873,A -85,B 0,C 180,E1 24589.824,E2 24589.824} C_VEL
LIN {X 0,Y 531.335,Z 631.837,A -85,B 0,C 180,E1 24588.6,E2 24588.6} C_VEL
LIN {X 0,Y 530.562,Z 646.088,A -85,B 0,C 180,E1 24587.271,E2 24587.271} C_VEL
LIN {X 0,Y 529.803,Z 659.701,A -85,B 0,C 180,E1 24585.742,E2 24585.742} C_VEL
LIN {X 0,Y 529.169,Z 671.804,A -85,B 0,C 180,E1 24584.107,E2 24584.107} C_VEL
LIN {X 0,Y 528.672,Z 682.608,A -85,B 0,C 180,E1 24582.34,E2 24582.34} C_VEL
LIN {X 0,Y 528.292,Z 691.95,A -85,B 0,C 180,E1 24580.468,E2 24580.468} C_VEL
LIN {X 0,Y 528.065,Z 699.796,A -85,B 0,C 180,E1 24578.493,E2 24578.493} C_VEL
LIN {X 0,Y 527.955,Z 706.594,A -85,B 0,C 180,E1 24576.306,E2 24576.306} C_VEL
LIN {X 0,Y 527.924,Z 710.997,A -85,B 0,C 180,E1 24574.345,E2 24574.345} C_VEL
LIN {X 0,Y 527.911,Z 713.744,A -85,B 0,C 180,E1 24572.388,E2 24572.388} C_VEL
LIN {X 0,Y 527.909,Z 714.927,A -85,B 0,C 180,E1 24570.326,E2 24570.326} C_VEL
LIN {X 0,Y 527.913,Z 714.374,A -85,B 0,C 180,E1 24568.264,E2 24568.264} C_VEL
LIN {X 0,Y 527.914,Z 712.226,A -85,B 0,C 180,E1 24566.308,E2 24566.308} C_VEL
LIN {X 0,Y 527.937,Z 708.455,A -85,B 0,C 180,E1 24564.348,E2 24564.348} C_VEL
LIN {X 0,Y 528.008,Z 702.639,A -85,B 0,C 180,E1 24562.274,E2 24562.274} C_VEL
LIN {X 0,Y 528.172,Z 695.607,A -85,B 0,C 180,E1 24560.301,E2 24560.301} C_VEL
LIN {X 0,Y 528.475,Z 687.161,A -85,B 0,C 180,E1 24558.431,E2 24558.431} C_VEL
LIN {X 0,Y 528.915,Z 677.344,A -85,B 0,C 180,E1 24556.666,E2 24556.666} C_VEL
LIN {X 0,Y 529.452,Z 666.189,A -85,B 0,C 180,E1 24555.006,E2 24555.006} C_VEL
LIN {X 0,Y 530.138,Z 653.641,A -85,B 0,C 180,E1 24553.454,E2 24553.454} C_VEL
LIN {X 0,Y 530.911,Z 639.573,A -85,B 0,C 180,E1 24552.002,E2 24552.002} C_VEL
LIN {X 0,Y 531.708,Z 624.712,A -85,B 0,C 180,E1 24550.734,E2 24550.734} C_VEL
LIN {X 0,Y 532.497,Z 608.695,A -85,B 0,C 180,E1 24549.617,E2 24549.617} C_VEL
LIN {X 0,Y 533.226,Z 591.689,A -85,B 0,C 180,E1 24548.669,E2 24548.669} C_VEL
LIN {X 0,Y 533.817,Z 574.117,A -85,B 0,C 180,E1 24547.914,E2 24547.914} C_VEL
LIN {X 0,Y 534.248,Z 555.617,A -85,B 0,C 180,E1 24547.338,E2 24547.338} C_VEL
LIN {X 0,Y 534.478,Z 536.527,A -85,B 0,C 180,E1 24546.962,E2 24546.962} C_VEL
LIN {X 0,Y 535.554,Z 346.222,A -85,B 0,C 180,E1 24544.316,E2 24544.316} C_VEL
LIN {X 0,Y 533.396,Z 336.077,A -85,B 0,C 180,E1 24544.011,E2 24544.011} C_VEL
LIN {X 0,Y 534.104,Z 313.814,A -85,B 0,C 180,E1 24541.852,E2 24541.852} C_VEL
LIN {X 0,Y 528.55,Z 296.845,A -85,B 0,C 180,E1 24539.664,E2 24539.664} C_VEL
LIN {X 0,Y 528.521,Z 296.638,A -85,B 0,C 180,E1 24536.208,E2 24536.208} C_VEL
LIN {X 0,Y 528.499,Z 296.648,A -85,B 0,C 180,E1 24532.796,E2 24532.796} C_VEL
LIN {X 0,Y 528.496,Z 296.654,A -85,B 0,C 180,E1 24529.256,E2 24529.256} C_VEL
LIN {X 0,Y 528.523,Z 296.631,A -85,B 0,C 180,E1 24525.807,E2 24525.807} C_VEL
LIN {X 0,Y 528.504,Z 296.649,A -85,B 0,C 180,E1 24522.455,E2 24522.455} C_VEL
LIN {X 0,Y 528.485,Z 296.651,A -85,B 0,C 180,E1 24519.051,E2 24519.051} C_VEL
LIN {X 0,Y 528.522,Z 296.654,A -85,B 0,C 180,E1 24515.639,E2 24515.639} C_VEL
LIN {X 0,Y 528.503,Z 296.648,A -85,B 0,C 180,E1 24512.243,E2 24512.243} C_VEL
LIN {X 0,Y 528.475,Z 296.65,A -85,B 0,C 180,E1 24508.97,E2 24508.97} C_VEL
LIN {X 0,Y 528.525,Z 296.647,A -85,B 0,C 180,E1 24505.672,E2 24505.672} C_VEL
LIN {X 0,Y 528.48,Z 296.652,A -85,B 0,C 180,E1 24502.311,E2 24502.311} C_VEL
LIN {X 0,Y 528.463,Z 296.65,A -85,B 0,C 180,E1 24498.877,E2 24498.877} C_VEL
LIN {X 0,Y 528.522,Z 296.648,A -85,B 0,C 180,E1 24495.583,E2 24495.583} C_VEL
LIN {X 0,Y 528.46,Z 296.652,A -85,B 0,C 180,E1 24492.345,E2 24492.345} C_VEL
LIN {X 0,Y 528.455,Z 296.645,A -85,B 0,C 180,E1 24488.816,E2 24488.816} C_VEL
LIN {X 0,Y 528.515,Z 296.655,A -85,B 0,C 180,E1 24485.537,E2 24485.537} C_VEL
LIN {X 0,Y 528.448,Z 296.647,A -85,B 0,C 180,E1 24482.277,E2 24482.277} C_VEL
LIN {X 0,Y 528.449,Z 296.652,A -85,B 0,C 180,E1 24478.808,E2 24478.808} C_VEL
LIN {X 0,Y 528.507,Z 296.65,A -85,B 0,C 180,E1 24475.545,E2 24475.545} C_VEL
LIN {X 0,Y 528.45,Z 296.649,A -85,B 0,C 180,E1 24472.28,E2 24472.28} C_VEL
LIN {X 0,Y 528.473,Z 296.653,A -85,B 0,C 180,E1 24468.873,E2 24468.873} C_VEL
LIN {X 0,Y 528.501,Z 296.646,A -85,B 0,C 180,E1 24465.607,E2 24465.607} C_VEL
LIN {X 0,Y 528.46,Z 296.65,A -85,B 0,C 180,E1 24462.379,E2 24462.379} C_VEL
LIN {X 0,Y 528.512,Z 296.65,A -85,B 0,C 180,E1 24459.05,E2 24459.05} C_VEL
LIN {X 0,Y 528.486,Z 296.65,A -85,B 0,C 180,E1 24455.767,E2 24455.767} C_VEL
LIN {X 0,Y 528.472,Z 296.648,A -85,B 0,C 180,E1 24452.385,E2 24452.385} C_VEL
LIN {X 0,Y 528.524,Z 296.646,A -85,B 0,C 180,E1 24449.032,E2 24449.032} C_VEL
LIN {X 0,Y 528.493,Z 296.649,A -85,B 0,C 180,E1 24445.682,E2 24445.682} C_VEL
LIN {X 0,Y 528.482,Z 296.647,A -85,B 0,C 180,E1 24442.261,E2 24442.261} C_VEL
LIN {X 0,Y 528.528,Z 296.63,A -85,B 0,C 180,E1 24438.971,E2 24438.971} C_VEL
LIN {X 0,Y 528.51,Z 296.654,A -85,B 0,C 180,E1 24435.496,E2 24435.496} C_VEL
LIN {X 0,Y 528.491,Z 296.653,A -85,B 0,C 180,E1 24432.045,E2 24432.045} C_VEL
LIN {X 0,Y 528.527,Z 296.642,A -85,B 0,C 180,E1 24428.767,E2 24428.767} C_VEL
LIN {X 0,Y 528.542,Z 296.967,A -85,B 0,C 180,E1 24428.178,E2 24428.178} C_VEL
LIN {X 0,Y 530.603,Z 302.33,A -85,B 0,C 180,E1 24427.627,E2 24427.627} C_VEL
LIN {X 0,Y 537.847,Z 320.134,A -85,B 0,C 180,E1 24425.975,E2 24425.975} C_VEL
LIN {X 0,Y 536.51,Z 373.681,A -85,B 0,C 180,E1 24422.713,E2 24422.713} C_VEL
LIN {X 0,Y 536.214,Z 390.662,A -85,B 0,C 180,E1 24421.726,E2 24421.726} C_VEL
LIN {X 0,Y 537.859,Z 403.647,A -85,B 0,C 180,E1 24421.434,E2 24421.434} C_VEL
LIN {X 0,Y 536.406,Z 594.787,A -85,B 0,C 180,E1 24418.683,E2 24418.683} C_VEL
LIN {X 0,Y 535.833,Z 654.415,A -85,B 0,C 180,E1 24417.791,E2 24417.791} C_VEL
LIN {X 0,Y 535.306,Z 675.429,A -85,B 0,C 180,E1 24417.273,E2 24417.273} C_VEL
LIN {X 0,Y 534.649,Z 695.21,A -85,B 0,C 180,E1 24416.581,E2 24416.581} C_VEL
LIN {X 0,Y 533.887,Z 714.635,A -85,B 0,C 180,E1 24415.698,E2 24415.698} C_VEL
LIN {X 0,Y 533.019,Z 733.838,A -85,B 0,C 180,E1 24414.609,E2 24414.609} C_VEL
LIN {X 0,Y 532.156,Z 751.982,A -85,B 0,C 180,E1 24413.355,E2 24413.355} C_VEL
LIN {X 0,Y 531.341,Z 768.574,A -85,B 0,C 180,E1 24411.991,E2 24411.991} C_VEL
LIN {X 0,Y 530.496,Z 785.443,A -85,B 0,C 180,E1 24410.341,E2 24410.341} C_VEL
LIN {X 0,Y 529.771,Z 800.448,A -85,B 0,C 180,E1 24408.599,E2 24408.599} C_VEL
LIN {X 0,Y 529.181,Z 813.584,A -85,B 0,C 180,E1 24406.803,E2 24406.803} C_VEL
LIN {X 0,Y 528.719,Z 825.381,A -85,B 0,C 180,E1 24404.903,E2 24404.903} C_VEL
LIN {X 0,Y 528.359,Z 836.336,A -85,B 0,C 180,E1 24402.791,E2 24402.791} C_VEL
LIN {X 0,Y 528.139,Z 845.251,A -85,B 0,C 180,E1 24400.692,E2 24400.692} C_VEL
LIN {X 0,Y 528.009,Z 852.377,A -85,B 0,C 180,E1 24398.603,E2 24398.603} C_VEL
LIN {X 0,Y 527.937,Z 858.005,A -85,B 0,C 180,E1 24396.415,E2 24396.415} C_VEL
LIN {X 0,Y 527.911,Z 861.929,A -85,B 0,C 180,E1 24394.236,E2 24394.236} C_VEL
LIN {X 0,Y 527.911,Z 864.306,A -85,B 0,C 180,E1 24391.954,E2 24391.954} C_VEL
LIN {X 0,Y 527.906,Z 864.962,A -85,B 0,C 180,E1 24389.783,E2 24389.783} C_VEL
LIN {X 0,Y 527.902,Z 864.033,A -85,B 0,C 180,E1 24387.612,E2 24387.612} C_VEL
LIN {X 0,Y 527.911,Z 861.449,A -85,B 0,C 180,E1 24385.438,E2 24385.438} C_VEL
LIN {X 0,Y 527.952,Z 857.245,A -85,B 0,C 180,E1 24383.257,E2 24383.257} C_VEL
LIN {X 0,Y 528.024,Z 851.327,A -85,B 0,C 180,E1 24381.068,E2 24381.068} C_VEL
LIN {X 0,Y 528.162,Z 844.013,A -85,B 0,C 180,E1 24378.977,E2 24378.977} C_VEL
LIN {X 0,Y 528.408,Z 834.783,A -85,B 0,C 180,E1 24376.876,E2 24376.876} C_VEL
LIN {X 0,Y 528.767,Z 824.109,A -85,B 0,C 180,E1 24374.874,E2 24374.874} C_VEL
LIN {X 0,Y 529.252,Z 811.725,A -85,B 0,C 180,E1 24372.926,E2 24372.926} C_VEL
LIN {X 0,Y 529.883,Z 797.67,A -85,B 0,C 180,E1 24371.062,E2 24371.062} C_VEL
LIN {X 0,Y 530.612,Z 782.615,A -85,B 0,C 180,E1 24369.368,E2 24369.368} C_VEL
LIN {X 0,Y 531.432,Z 766.62,A -85,B 0,C 180,E1 24367.839,E2 24367.839} C_VEL
LIN {X 0,Y 532.325,Z 748.992,A -85,B 0,C 180,E1 24366.418,E2 24366.418} C_VEL
LIN {X 0,Y 533.204,Z 730.23,A -85,B 0,C 180,E1 24365.164,E2 24365.164} C_VEL
LIN {X 0,Y 534.017,Z 711.348,A -85,B 0,C 180,E1 24364.136,E2 24364.136} C_VEL
LIN {X 0,Y 534.758,Z 692.224,A -85,B 0,C 180,E1 24363.304,E2 24363.304} C_VEL
LIN {X 0,Y 535.382,Z 671.626,A -85,B 0,C 180,E1 24362.621,E2 24362.621} C_VEL
LIN {X 0,Y 535.881,Z 651.072,A -85,B 0,C 180,E1 24362.149,E2 24362.149} C_VEL
LIN {X 0,Y 537.542,Z 449.728,A -85,B 0,C 180,E1 24359.224,E2 24359.224} C_VEL
LIN {X 0,Y 537.667,Z 400.554,A -85,B 0,C 180,E1 24358.508,E2 24358.508} C_VEL
LIN {X 0,Y 536.131,Z 389.177,A -85,B 0,C 180,E1 24358.215,E2 24358.215} C_VEL
LIN {X 0,Y 537.478,Z 334.555,A -85,B 0,C 180,E1 24354.914,E2 24354.914} C_VEL
LIN {X 0,Y 537.765,Z 319.473,A -85,B 0,C 180,E1 24353.977,E2 24353.977} C_VEL
LIN {X 0,Y 528.559,Z 297.071,A -85,B 0,C 180,E1 24351.843,E2 24351.843} C_VEL
LIN {X 0,Y 528.513,Z 296.65,A -85,B 0,C 180,E1 24351.509,E2 24351.509} C_VEL
LIN {X 0,Y 528.491,Z 296.654,A -85,B 0,C 180,E1 24348.101,E2 24348.101} C_VEL
LIN {X 0,Y 528.521,Z 296.649,A -85,B 0,C 180,E1 24344.659,E2 24344.659} C_VEL
LIN {X 0,Y 528.524,Z 296.628,A -85,B 0,C 180,E1 24341.173,E2 24341.173} C_VEL
LIN {X 0,Y 528.482,Z 296.647,A -85,B 0,C 180,E1 24337.806,E2 24337.806} C_VEL
LIN {X 0,Y 528.504,Z 296.645,A -85,B 0,C 180,E1 24334.429,E2 24334.429} C_VEL
LIN {X 0,Y 528.514,Z 296.647,A -85,B 0,C 180,E1 24331.095,E2 24331.095} C_VEL
LIN {X 0,Y 528.473,Z 296.648,A -85,B 0,C 180,E1 24327.738,E2 24327.738} C_VEL
LIN {X 0,Y 528.5,Z 296.651,A -85,B 0,C 180,E1 24324.357,E2 24324.357} C_VEL
LIN {X 0,Y 528.492,Z 296.651,A -85,B 0,C 180,E1 24321.143,E2 24321.143} C_VEL
LIN {X 0,Y 528.463,Z 296.65,A -85,B 0,C 180,E1 24317.735,E2 24317.735} C_VEL
LIN {X 0,Y 528.505,Z 296.646,A -85,B 0,C 180,E1 24314.395,E2 24314.395} C_VEL
LIN {X 0,Y 528.474,Z 296.652,A -85,B 0,C 180,E1 24311.127,E2 24311.127} C_VEL
LIN {X 0,Y 528.454,Z 296.649,A -85,B 0,C 180,E1 24307.72,E2 24307.72} C_VEL
LIN {X 0,Y 528.511,Z 296.651,A -85,B 0,C 180,E1 24304.448,E2 24304.448} C_VEL
LIN {X 0,Y 528.453,Z 296.652,A -85,B 0,C 180,E1 24301.192,E2 24301.192} C_VEL
LIN {X 0,Y 528.445,Z 296.648,A -85,B 0,C 180,E1 24297.723,E2 24297.723} C_VEL
LIN {X 0,Y 528.509,Z 296.654,A -85,B 0,C 180,E1 24294.463,E2 24294.463} C_VEL
LIN {X 0,Y 528.446,Z 296.645,A -85,B 0,C 180,E1 24291.294,E2 24291.294} C_VEL
LIN {X 0,Y 528.481,Z 296.652,A -85,B 0,C 180,E1 24287.988,E2 24287.988} C_VEL
LIN {X 0,Y 528.469,Z 296.647,A -85,B 0,C 180,E1 24284.865,E2 24284.865} C_VEL
LIN {X 0,Y 528.46,Z 296.649,A -85,B 0,C 180,E1 24281.419,E2 24281.419} C_VEL
LIN {X 0,Y 528.519,Z 296.651,A -85,B 0,C 180,E1 24278.118,E2 24278.118} C_VEL
LIN {X 0,Y 528.476,Z 296.646,A -85,B 0,C 180,E1 24274.805,E2 24274.805} C_VEL
LIN {X 0,Y 528.471,Z 296.649,A -85,B 0,C 180,E1 24271.385,E2 24271.385} C_VEL
LIN {X 0,Y 528.53,Z 296.651,A -85,B 0,C 180,E1 24268.142,E2 24268.142} C_VEL
LIN {X 0,Y 528.482,Z 296.652,A -85,B 0,C 180,E1 24264.757,E2 24264.757} C_VEL
LIN {X 0,Y 528.507,Z 296.648,A -85,B 0,C 180,E1 24261.691,E2 24261.691} C_VEL
LIN {X 0,Y 527.481,Z 296.777,A -85,B 0,C 180,E1 24260.857,E2 24260.857} C_VEL
LIN {X 0,Y 521.034,Z 297.584,A -85,B 0,C 180,E1 24258.45,E2 24258.45} C_VEL
LIN {X 0,Y 520.588,Z 297.638,A -85,B 0,C 180,E1 24257.9,E2 24257.9} C_VEL
LIN {X 0,Y 520.562,Z 297.625,A -85,B 0,C 180,E1 24254.511,E2 24254.511} C_VEL
LIN {X 0,Y 520.548,Z 297.642,A -85,B 0,C 180,E1 24251.063,E2 24251.063} C_VEL
LIN {X 0,Y 520.582,Z 297.628,A -85,B 0,C 180,E1 24247.644,E2 24247.644} C_VEL
LIN {X 0,Y 520.583,Z 297.622,A -85,B 0,C 180,E1 24244.126,E2 24244.126} C_VEL
LIN {X 0,Y 520.579,Z 297.806,A -85,B 0,C 180,E1 24240.755,E2 24240.755} C_VEL
LIN {X 0,Y 526.918,Z 316.989,A -85,B 0,C 180,E1 24238.234,E2 24238.234} C_VEL
LIN {X 0,Y 526.229,Z 337.08,A -85,B 0,C 180,E1 24236.302,E2 24236.302} C_VEL
LIN {X 0,Y 528.672,Z 349.224,A -85,B 0,C 180,E1 24235.966,E2 24235.966} C_VEL
LIN {X 0,Y 527.369,Z 546.9,A -85,B 0,C 180,E1 24233.192,E2 24233.192} C_VEL
LIN {X 0,Y 527.036,Z 565.736,A -85,B 0,C 180,E1 24232.713,E2 24232.713} C_VEL
LIN {X 0,Y 526.49,Z 583.327,A -85,B 0,C 180,E1 24232.064,E2 24232.064} C_VEL
LIN {X 0,Y 525.813,Z 600.136,A -85,B 0,C 180,E1 24231.238,E2 24231.238} C_VEL
LIN {X 0,Y 524.982,Z 616.458,A -85,B 0,C 180,E1 24230.223,E2 24230.223} C_VEL
LIN {X 0,Y 524.076,Z 632.536,A -85,B 0,C 180,E1 24228.983,E2 24228.983} C_VEL
LIN {X 0,Y 523.164,Z 647.431,A -85,B 0,C 180,E1 24227.575,E2 24227.575} C_VEL
LIN {X 0,Y 522.291,Z 661.177,A -85,B 0,C 180,E1 24226.001,E2 24226.001} C_VEL
LIN {X 0,Y 521.551,Z 673.351,A -85,B 0,C 180,E1 24224.318,E2 24224.318} C_VEL
LIN {X 0,Y 520.971,Z 684.051,A -85,B 0,C 180,E1 24222.525,E2 24222.525} C_VEL
LIN {X 0,Y 520.525,Z 693.329,A -85,B 0,C 180,E1 24220.626,E2 24220.626} C_VEL
LIN {X 0,Y 520.241,Z 701.12,A -85,B 0,C 180,E1 24218.621,E2 24218.621} C_VEL
LIN {X 0,Y 520.062,Z 707.368,A -85,B 0,C 180,E1 24216.513,E2 24216.513} C_VEL
LIN {X 0,Y 519.972,Z 711.771,A -85,B 0,C 180,E1 24214.411,E2 24214.411} C_VEL
LIN {X 0,Y 519.937,Z 714.447,A -85,B 0,C 180,E1 24212.314,E2 24212.314} C_VEL
LIN {X 0,Y 519.928,Z 715.468,A -85,B 0,C 180,E1 24210.22,E2 24210.22} C_VEL
LIN {X 0,Y 519.935,Z 714.863,A -85,B 0,C 180,E1 24208.127,E2 24208.127} C_VEL
LIN {X 0,Y 519.959,Z 712.615,A -85,B 0,C 180,E1 24206.031,E2 24206.031} C_VEL
LIN {X 0,Y 520.032,Z 708.67,A -85,B 0,C 180,E1 24203.93,E2 24203.93} C_VEL
LIN {X 0,Y 520.194,Z 702.925,A -85,B 0,C 180,E1 24201.823,E2 24201.823} C_VEL
LIN {X 0,Y 520.44,Z 695.647,A -85,B 0,C 180,E1 24199.82,E2 24199.82} C_VEL
LIN {X 0,Y 520.865,Z 686.322,A -85,B 0,C 180,E1 24197.81,E2 24197.81} C_VEL
LIN {X 0,Y 521.412,Z 675.998,A -85,B 0,C 180,E1 24196.003,E2 24196.003} C_VEL
LIN {X 0,Y 522.09,Z 664.479,A -85,B 0,C 180,E1 24194.334,E2 24194.334} C_VEL
LIN {X 0,Y 522.912,Z 651.395,A -85,B 0,C 180,E1 24192.761,E2 24192.761} C_VEL
LIN {X 0,Y 523.776,Z 637.316,A -85,B 0,C 180,E1 24191.353,E2 24191.353} C_VEL
LIN {X 0,Y 524.663,Z 622.309,A -85,B 0,C 180,E1 24190.113,E2 24190.113} C_VEL
LIN {X 0,Y 525.501,Z 606.44,A -85,B 0,C 180,E1 24189.041,E2 24189.041} C_VEL
LIN {X 0,Y 526.243,Z 589.686,A -85,B 0,C 180,E1 24188.137,E2 24188.137} C_VEL
LIN {X 0,Y 526.854,Z 572.11,A -85,B 0,C 180,E1 24187.411,E2 24187.411} C_VEL
LIN {X 0,Y 527.266,Z 553.957,A -85,B 0,C 180,E1 24186.875,E2 24186.875} C_VEL
LIN {X 0,Y 527.468,Z 534.429,A -85,B 0,C 180,E1 24186.515,E2 24186.515} C_VEL
LIN {X 0,Y 528.54,Z 347.505,A -85,B 0,C 180,E1 24183.91,E2 24183.91} C_VEL
LIN {X 0,Y 526.205,Z 336.939,A -85,B 0,C 180,E1 24183.601,E2 24183.601} C_VEL
LIN {X 0,Y 526.942,Z 317.05,A -85,B 0,C 180,E1 24181.683,E2 24181.683} C_VEL
LIN {X 0,Y 520.582,Z 297.802,A -85,B 0,C 180,E1 24179.15,E2 24179.15} C_VEL
LIN {X 0,Y 520.579,Z 297.622,A -85,B 0,C 180,E1 24175.679,E2 24175.679} C_VEL
LIN {X 0,Y 520.586,Z 297.627,A -85,B 0,C 180,E1 24172.217,E2 24172.217} C_VEL
LIN {X 0,Y 520.556,Z 297.64,A -85,B 0,C 180,E1 24168.792,E2 24168.792} C_VEL
LIN {X 0,Y 520.557,Z 297.627,A -85,B 0,C 180,E1 24165.29,E2 24165.29} C_VEL
LIN {X 0,Y 520.589,Z 297.638,A -85,B 0,C 180,E1 24161.942,E2 24161.942} C_VEL
LIN {X 0,Y 520.551,Z 297.637,A -85,B 0,C 180,E1 24158.581,E2 24158.581} C_VEL
LIN {X 0,Y 520.543,Z 297.639,A -85,B 0,C 180,E1 24155.052,E2 24155.052} C_VEL
LIN {X 0,Y 520.585,Z 297.643,A -85,B 0,C 180,E1 24151.624,E2 24151.624} C_VEL
LIN {X 0,Y 520.552,Z 297.636,A -85,B 0,C 180,E1 24148.323,E2 24148.323} C_VEL
LIN {X 0,Y 520.53,Z 297.633,A -85,B 0,C 180,E1 24144.877,E2 24144.877} C_VEL
LIN {X 0,Y 520.578,Z 297.64,A -85,B 0,C 180,E1 24141.522,E2 24141.522} C_VEL
LIN {X 0,Y 520.538,Z 297.637,A -85,B 0,C 180,E1 24138.246,E2 24138.246} C_VEL
LIN {X 0,Y 520.519,Z 297.634,A -85,B 0,C 180,E1 24134.802,E2 24134.802} C_VEL
LIN {X 0,Y 520.576,Z 297.644,A -85,B 0,C 180,E1 24131.523,E2 24131.523} C_VEL
LIN {X 0,Y 520.524,Z 297.632,A -85,B 0,C 180,E1 24128.172,E2 24128.172} C_VEL
LIN {X 0,Y 520.51,Z 297.642,A -85,B 0,C 180,E1 24124.738,E2 24124.738} C_VEL
LIN {X 0,Y 520.568,Z 297.638,A -85,B 0,C 180,E1 24121.431,E2 24121.431} C_VEL
LIN {X 0,Y 520.513,Z 297.64,A -85,B 0,C 180,E1 24118.129,E2 24118.129} C_VEL
LIN {X 0,Y 520.513,Z 297.643,A -85,B 0,C 180,E1 24114.71,E2 24114.71} C_VEL
LIN {X 0,Y 520.573,Z 297.633,A -85,B 0,C 180,E1 24111.495,E2 24111.495} C_VEL
LIN {X 0,Y 520.52,Z 297.643,A -85,B 0,C 180,E1 24108.139,E2 24108.139} C_VEL
LIN {X 0,Y 520.526,Z 297.642,A -85,B 0,C 180,E1 24104.629,E2 24104.629} C_VEL
LIN {X 0,Y 520.583,Z 297.634,A -85,B 0,C 180,E1 24101.292,E2 24101.292} C_VEL
LIN {X 0,Y 520.532,Z 297.642,A -85,B 0,C 180,E1 24098.003,E2 24098.003} C_VEL
LIN {X 0,Y 520.536,Z 297.641,A -85,B 0,C 180,E1 24094.516,E2 24094.516} C_VEL
LIN {X 0,Y 520.589,Z 297.64,A -85,B 0,C 180,E1 24091.137,E2 24091.137} C_VEL
LIN {X 0,Y 520.551,Z 297.641,A -85,B 0,C 180,E1 24087.726,E2 24087.726} C_VEL
LIN {X 0,Y 520.539,Z 297.621,A -85,B 0,C 180,E1 24084.273,E2 24084.273} C_VEL
LIN {X 0,Y 520.589,Z 297.637,A -85,B 0,C 180,E1 24080.888,E2 24080.888} C_VEL
LIN {X 0,Y 520.572,Z 297.622,A -85,B 0,C 180,E1 24077.462,E2 24077.462} C_VEL
LIN {X 0,Y 520.548,Z 297.626,A -85,B 0,C 180,E1 24074.051,E2 24074.051} C_VEL
LIN {X 0,Y 520.584,Z 297.625,A -85,B 0,C 180,E1 24070.623,E2 24070.623} C_VEL
LIN {X 0,Y 520.602,Z 297.735,A -85,B 0,C 180,E1 24068.762,E2 24068.762} C_VEL
LIN {X 0,Y 520.932,Z 299.194,A -85,B 0,C 180,E1 24068.552,E2 24068.552} C_VEL
LIN {X 0,Y 530.761,Z 322.797,A -85,B 0,C 180,E1 24066.278,E2 24066.278} C_VEL
LIN {X 0,Y 529.242,Z 376.53,A -85,B 0,C 180,E1 24062.962,E2 24062.962} C_VEL
LIN {X 0,Y 528.955,Z 390.189,A -85,B 0,C 180,E1 24062.157,E2 24062.157} C_VEL
LIN {X 0,Y 530.787,Z 404.692,A -85,B 0,C 180,E1 24061.824,E2 24061.824} C_VEL
LIN {X 0,Y 529.1,Z 621.359,A -85,B 0,C 180,E1 24058.704,E2 24058.704} C_VEL
LIN {X 0,Y 528.723,Z 655.388,A -85,B 0,C 180,E1 24058.175,E2 24058.175} C_VEL
LIN {X 0,Y 528.15,Z 676.307,A -85,B 0,C 180,E1 24057.647,E2 24057.647} C_VEL
LIN {X 0,Y 527.422,Z 696.021,A -85,B 0,C 180,E1 24056.941,E2 24056.941} C_VEL
LIN {X 0,Y 526.599,Z 714.743,A -85,B 0,C 180,E1 24056.074,E2 24056.074} C_VEL
LIN {X 0,Y 525.642,Z 733.835,A -85,B 0,C 180,E1 24054.978,E2 24054.978} C_VEL
LIN {X 0,Y 524.69,Z 751.979,A -85,B 0,C 180,E1 24053.708,E2 24053.708} C_VEL
LIN {X 0,Y 523.737,Z 769.18,A -85,B 0,C 180,E1 24052.268,E2 24052.268} C_VEL
LIN {X 0,Y 522.831,Z 785.377,A -85,B 0,C 180,E1 24050.66,E2 24050.66} C_VEL
LIN {X 0,Y 522.011,Z 800.505,A -85,B 0,C 180,E1 24048.879,E2 24048.879} C_VEL
LIN {X 0,Y 521.319,Z 814.353,A -85,B 0,C 180,E1 24046.949,E2 24046.949} C_VEL
LIN {X 0,Y 520.807,Z 826.015,A -85,B 0,C 180,E1 24045.021,E2 24045.021} C_VEL
LIN {X 0,Y 520.406,Z 836.85,A -85,B 0,C 180,E1 24042.877,E2 24042.877} C_VEL
LIN {X 0,Y 520.152,Z 846.063,A -85,B 0,C 180,E1 24040.634,E2 24040.634} C_VEL
LIN {X 0,Y 520.008,Z 853.292,A -85,B 0,C 180,E1 24038.403,E2 24038.403} C_VEL
LIN {X 0,Y 519.941,Z 858.728,A -85,B 0,C 180,E1 24036.182,E2 24036.182} C_VEL
LIN {X 0,Y 519.916,Z 862.403,A -85,B 0,C 180,E1 24033.97,E2 24033.97} C_VEL
LIN {X 0,Y 519.907,Z 864.442,A -85,B 0,C 180,E1 24031.763,E2 24031.763} C_VEL
LIN {X 0,Y 519.9,Z 864.895,A -85,B 0,C 180,E1 24029.449,E2 24029.449} C_VEL
LIN {X 0,Y 519.912,Z 863.73,A -85,B 0,C 180,E1 24027.244,E2 24027.244} C_VEL
LIN {X 0,Y 519.93,Z 860.86,A -85,B 0,C 180,E1 24024.967,E2 24024.967} C_VEL
LIN {X 0,Y 519.971,Z 856.228,A -85,B 0,C 180,E1 24022.709,E2 24022.709} C_VEL
LIN {X 0,Y 520.067,Z 850.267,A -85,B 0,C 180,E1 24020.595,E2 24020.595} C_VEL
LIN {X 0,Y 520.251,Z 842.178,A -85,B 0,C 180,E1 24018.358,E2 24018.358} C_VEL
LIN {X 0,Y 520.563,Z 832.564,A -85,B 0,C 180,E1 24016.222,E2 24016.222} C_VEL
LIN {X 0,Y 521.001,Z 821.489,A -85,B 0,C 180,E1 24014.187,E2 24014.187} C_VEL
LIN {X 0,Y 521.587,Z 808.952,A -85,B 0,C 180,E1 24012.255,E2 24012.255} C_VEL
LIN {X 0,Y 522.304,Z 794.891,A -85,B 0,C 180,E1 24010.428,E2 24010.428} C_VEL
LIN {X 0,Y 523.127,Z 779.839,A -85,B 0,C 180,E1 24008.766,E2 24008.766} C_VEL
LIN {X 0,Y 524.048,Z 763.286,A -85,B 0,C 180,E1 24007.213,E2 24007.213} C_VEL
LIN {X 0,Y 525.059,Z 745.028,A -85,B 0,C 180,E1 24005.779,E2 24005.779} C_VEL
LIN {X 0,Y 526.045,Z 726.288,A -85,B 0,C 180,E1 24004.561,E2 24004.561} C_VEL
LIN {X 0,Y 526.947,Z 707.342,A -85,B 0,C 180,E1 24003.557,E2 24003.557} C_VEL
LIN {X 0,Y 527.74,Z 687.885,A -85,B 0,C 180,E1 24002.741,E2 24002.741} C_VEL
LIN {X 0,Y 528.402,Z 667.723,A -85,B 0,C 180,E1 24002.114,E2 24002.114} C_VEL
LIN {X 0,Y 528.851,Z 647.19,A -85,B 0,C 180,E1 24001.676,E2 24001.676} C_VEL
LIN {X 0,Y 530.711,Z 411.968,A -85,B 0,C 180,E1 23998.284,E2 23998.284} C_VEL
LIN {X 0,Y 530.565,Z 401.444,A -85,B 0,C 180,E1 23998.113,E2 23998.113} C_VEL
LIN {X 0,Y 528.878,Z 388.739,A -85,B 0,C 180,E1 23997.784,E2 23997.784} C_VEL
LIN {X 0,Y 530.436,Z 334.357,A -85,B 0,C 180,E1 23994.444,E2 23994.444} C_VEL
LIN {X 0,Y 530.669,Z 322.582,A -85,B 0,C 180,E1 23993.701,E2 23993.701} C_VEL
LIN {X 0,Y 520.651,Z 298.067,A -85,B 0,C 180,E1 23991.319,E2 23991.319} C_VEL
LIN {X 0,Y 520.584,Z 297.624,A -85,B 0,C 180,E1 23990.953,E2 23990.953} C_VEL
LIN {X 0,Y 520.568,Z 297.635,A -85,B 0,C 180,E1 23987.523,E2 23987.523} C_VEL
LIN {X 0,Y 520.549,Z 297.643,A -85,B 0,C 180,E1 23984.053,E2 23984.053} C_VEL
LIN {X 0,Y 520.582,Z 297.625,A -85,B 0,C 180,E1 23980.624,E2 23980.624} C_VEL
LIN {X 0,Y 520.581,Z 297.626,A -85,B 0,C 180,E1 23977.151,E2 23977.151} C_VEL
LIN {X 0,Y 520.541,Z 297.64,A -85,B 0,C 180,E1 23973.718,E2 23973.718} C_VEL
LIN {X 0,Y 520.55,Z 297.644,A -85,B 0,C 180,E1 23970.214,E2 23970.214} C_VEL
LIN {X 0,Y 520.581,Z 297.634,A -85,B 0,C 180,E1 23966.954,E2 23966.954} C_VEL
LIN {X 0,Y 520.531,Z 297.637,A -85,B 0,C 180,E1 23963.621,E2 23963.621} C_VEL
LIN {X 0,Y 520.549,Z 297.641,A -85,B 0,C 180,E1 23960.227,E2 23960.227} C_VEL
LIN {X 0,Y 520.572,Z 297.637,A -85,B 0,C 180,E1 23956.859,E2 23956.859} C_VEL
LIN {X 0,Y 520.519,Z 297.632,A -85,B 0,C 180,E1 23953.553,E2 23953.553} C_VEL
LIN {X 0,Y 520.544,Z 297.641,A -85,B 0,C 180,E1 23950.178,E2 23950.178} C_VEL
LIN {X 0,Y 520.542,Z 297.637,A -85,B 0,C 180,E1 23946.95,E2 23946.95} C_VEL
LIN {X 0,Y 520.51,Z 297.638,A -85,B 0,C 180,E1 23943.634,E2 23943.634} C_VEL
LIN {X 0,Y 520.563,Z 297.644,A -85,B 0,C 180,E1 23940.33,E2 23940.33} C_VEL
LIN {X 0,Y 520.516,Z 297.636,A -85,B 0,C 180,E1 23937.027,E2 23937.027} C_VEL
LIN {X 0,Y 520.508,Z 297.643,A -85,B 0,C 180,E1 23933.603,E2 23933.603} C_VEL
LIN {X 0,Y 520.572,Z 297.635,A -85,B 0,C 180,E1 23930.381,E2 23930.381} C_VEL
LIN {X 0,Y 520.516,Z 297.642,A -85,B 0,C 180,E1 23927.125,E2 23927.125} C_VEL
LIN {X 0,Y 520.524,Z 297.642,A -85,B 0,C 180,E1 23923.598,E2 23923.598} C_VEL
LIN {X 0,Y 520.581,Z 297.632,A -85,B 0,C 180,E1 23920.236,E2 23920.236} C_VEL
LIN {X 0,Y 520.531,Z 297.643,A -85,B 0,C 180,E1 23916.93,E2 23916.93} C_VEL
LIN {X 0,Y 520.531,Z 297.641,A -85,B 0,C 180,E1 23913.413,E2 23913.413} C_VEL
LIN {X 0,Y 520.591,Z 297.634,A -85,B 0,C 180,E1 23910.042,E2 23910.042} C_VEL
LIN {X 0,Y 520.551,Z 297.642,A -85,B 0,C 180,E1 23906.669,E2 23906.669} C_VEL
LIN {X 0,Y 520.538,Z 297.641,A -85,B 0,C 180,E1 23903.18,E2 23903.18} C_VEL
LIN {X 0,Y 520.58,Z 297.637,A -85,B 0,C 180,E1 23899.808,E2 23899.808} C_VEL
LIN {X 0,Y 520.588,Z 297.638,A -85,B 0,C 180,E1 23897.9,E2 23897.9} C_VEL
LIN {X 0,Y 519.576,Z 297.762,A -85,B 0,C 180,E1 23897.052,E2 23897.052} C_VEL
LIN {X 0,Y 513.168,Z 298.548,A -85,B 0,C 180,E1 23894.67,E2 23894.67} C_VEL
LIN {X 0,Y 512.646,Z 298.604,A -85,B 0,C 180,E1 23894.05,E2 23894.05} C_VEL
LIN {X 0,Y 512.616,Z 298.634,A -85,B 0,C 180,E1 23890.646,E2 23890.646} C_VEL
LIN {X 0,Y 512.614,Z 298.627,A -85,B 0,C 180,E1 23887.083,E2 23887.083} C_VEL
LIN {X 0,Y 512.644,Z 298.613,A -85,B 0,C 180,E1 23883.61,E2 23883.61} C_VEL
LIN {X 0,Y 512.665,Z 298.875,A -85,B 0,C 180,E1 23881.25,E2 23881.25} C_VEL
LIN {X 0,Y 519.539,Z 319.478,A -85,B 0,C 180,E1 23878.507,E2 23878.507} C_VEL
LIN {X 0,Y 519.024,Z 337.459,A -85,B 0,C 180,E1 23876.752,E2 23876.752} C_VEL
LIN {X 0,Y 521.699,Z 350.573,A -85,B 0,C 180,E1 23876.38,E2 23876.38} C_VEL
LIN {X 0,Y 520.375,Z 547.955,A -85,B 0,C 180,E1 23873.604,E2 23873.604} C_VEL
LIN {X 0,Y 520.037,Z 566.771,A -85,B 0,C 180,E1 23873.122,E2 23873.122} C_VEL
LIN {X 0,Y 519.458,Z 584.493,A -85,B 0,C 180,E1 23872.462,E2 23872.462} C_VEL
LIN {X 0,Y 518.708,Z 601.722,A -85,B 0,C 180,E1 23871.602,E2 23871.602} C_VEL
LIN {X 0,Y 517.807,Z 617.966,A -85,B 0,C 180,E1 23870.574,E2 23870.574} C_VEL
LIN {X 0,Y 516.804,Z 633.932,A -85,B 0,C 180,E1 23869.319,E2 23869.319} C_VEL
LIN {X 0,Y 515.83,Z 648.22,A -85,B 0,C 180,E1 23867.95,E2 23867.95} C_VEL
LIN {X 0,Y 514.848,Z 661.999,A -85,B 0,C 180,E1 23866.355,E2 23866.355} C_VEL
LIN {X 0,Y 514.002,Z 674.218,A -85,B 0,C 180,E1 23864.648,E2 23864.648} C_VEL
LIN {X 0,Y 513.328,Z 684.954,A -85,B 0,C 180,E1 23862.829,E2 23862.829} C_VEL
LIN {X 0,Y 512.79,Z 694.248,A -85,B 0,C 180,E1 23860.902,E2 23860.902} C_VEL
LIN {X 0,Y 512.43,Z 702.067,A -85,B 0,C 180,E1 23858.867,E2 23858.867} C_VEL
LIN {X 0,Y 512.211,Z 708.354,A -85,B 0,C 180,E1 23856.726,E2 23856.726} C_VEL
LIN {X 0,Y 512.086,Z 712.811,A -85,B 0,C 180,E1 23854.592,E2 23854.592} C_VEL
LIN {X 0,Y 512.031,Z 715.552,A -85,B 0,C 180,E1 23852.462,E2 23852.462} C_VEL
LIN {X 0,Y 512.018,Z 716.649,A -85,B 0,C 180,E1 23850.336,E2 23850.336} C_VEL
LIN {X 0,Y 512.027,Z 716.132,A -85,B 0,C 180,E1 23848.21,E2 23848.21} C_VEL
LIN {X 0,Y 512.061,Z 713.989,A -85,B 0,C 180,E1 23846.081,E2 23846.081} C_VEL
LIN {X 0,Y 512.153,Z 710.161,A -85,B 0,C 180,E1 23843.949,E2 23843.949} C_VEL
LIN {X 0,Y 512.346,Z 704.552,A -85,B 0,C 180,E1 23841.81,E2 23841.81} C_VEL
LIN {X 0,Y 512.637,Z 697.451,A -85,B 0,C 180,E1 23839.777,E2 23839.777} C_VEL
LIN {X 0,Y 513.133,Z 688.386,A -85,B 0,C 180,E1 23837.738,E2 23837.738} C_VEL
LIN {X 0,Y 513.787,Z 677.664,A -85,B 0,C 180,E1 23835.807,E2 23835.807} C_VEL
LIN {X 0,Y 514.558,Z 666.154,A -85,B 0,C 180,E1 23834.099,E2 23834.099} C_VEL
LIN {X 0,Y 515.475,Z 653.203,A -85,B 0,C 180,E1 23832.504,E2 23832.504} C_VEL
LIN {X 0,Y 516.437,Z 639.312,A -85,B 0,C 180,E1 23831.078,E2 23831.078} C_VEL
LIN {X 0,Y 517.416,Z 624.536,A -85,B 0,C 180,E1 23829.823,E2 23829.823} C_VEL
LIN {X 0,Y 518.326,Z 608.947,A -85,B 0,C 180,E1 23828.737,E2 23828.737} C_VEL
LIN {X 0,Y 519.137,Z 592.552,A -85,B 0,C 180,E1 23827.822,E2 23827.822} C_VEL
LIN {X 0,Y 519.815,Z 574.501,A -85,B 0,C 180,E1 23827.051,E2 23827.051} C_VEL
LIN {X 0,Y 520.26,Z 556.025,A -85,B 0,C 180,E1 23826.487,E2 23826.487} C_VEL
LIN {X 0,Y 520.461,Z 536.725,A -85,B 0,C 180,E1 23826.12,E2 23826.12} C_VEL
LIN {X 0,Y 521.552,Z 348.835,A -85,B 0,C 180,E1 23823.494,E2 23823.494} C_VEL
LIN {X 0,Y 518.981,Z 336.969,A -85,B 0,C 180,E1 23823.127,E2 23823.127} C_VEL
LIN {X 0,Y 519.601,Z 319.667,A -85,B 0,C 180,E1 23821.428,E2 23821.428} C_VEL
LIN {X 0,Y 513.355,Z 301.104,A -85,B 0,C 180,E1 23818.98,E2 23818.98} C_VEL
LIN {X 0,Y 512.658,Z 298.755,A -85,B 0,C 180,E1 23818.619,E2 23818.619} C_VEL
LIN {X 0,Y 512.618,Z 298.615,A -85,B 0,C 180,E1 23815.147,E2 23815.147} C_VEL
LIN {X 0,Y 512.64,Z 298.609,A -85,B 0,C 180,E1 23811.635,E2 23811.635} C_VEL
LIN {X 0,Y 512.65,Z 298.628,A -85,B 0,C 180,E1 23808.163,E2 23808.163} C_VEL
LIN {X 0,Y 512.614,Z 298.622,A -85,B 0,C 180,E1 23804.76,E2 23804.76} C_VEL
LIN {X 0,Y 512.614,Z 298.628,A -85,B 0,C 180,E1 23801.245,E2 23801.245} C_VEL
LIN {X 0,Y 512.65,Z 298.623,A -85,B 0,C 180,E1 23797.826,E2 23797.826} C_VEL
LIN {X 0,Y 512.617,Z 298.625,A -85,B 0,C 180,E1 23794.408,E2 23794.408} C_VEL
LIN {X 0,Y 512.6,Z 298.629,A -85,B 0,C 180,E1 23790.994,E2 23790.994} C_VEL
LIN {X 0,Y 512.646,Z 298.629,A -85,B 0,C 180,E1 23787.658,E2 23787.658} C_VEL
LIN {X 0,Y 512.606,Z 298.62,A -85,B 0,C 180,E1 23784.303,E2 23784.303} C_VEL
LIN {X 0,Y 512.591,Z 298.627,A -85,B 0,C 180,E1 23780.883,E2 23780.883} C_VEL
LIN {X 0,Y 512.633,Z 298.632,A -85,B 0,C 180,E1 23777.48,E2 23777.48} C_VEL
LIN {X 0,Y 512.601,Z 298.621,A -85,B 0,C 180,E1 23774.112,E2 23774.112} C_VEL
LIN {X 0,Y 512.576,Z 298.631,A -85,B 0,C 180,E1 23770.68,E2 23770.68} C_VEL
LIN {X 0,Y 512.612,Z 298.631,A -85,B 0,C 180,E1 23767.284,E2 23767.284} C_VEL
LIN {X 0,Y 512.589,Z 298.631,A -85,B 0,C 180,E1 23764.027,E2 23764.027} C_VEL
LIN {X 0,Y 512.566,Z 298.633,A -85,B 0,C 180,E1 23760.671,E2 23760.671} C_VEL
LIN {X 0,Y 512.628,Z 298.62,A -85,B 0,C 180,E1 23757.429,E2 23757.429} C_VEL
LIN {X 0,Y 512.581,Z 298.632,A -85,B 0,C 180,E1 23754.066,E2 23754.066} C_VEL
LIN {X 0,Y 512.576,Z 298.629,A -85,B 0,C 180,E1 23750.57,E2 23750.57} C_VEL
LIN {X 0,Y 512.632,Z 298.62,A -85,B 0,C 180,E1 23747.211,E2 23747.211} C_VEL
LIN {X 0,Y 512.594,Z 298.632,A -85,B 0,C 180,E1 23743.92,E2 23743.92} C_VEL
LIN {X 0,Y 512.587,Z 298.628,A -85,B 0,C 180,E1 23740.41,E2 23740.41} C_VEL
LIN {X 0,Y 512.637,Z 298.622,A -85,B 0,C 180,E1 23737.04,E2 23737.04} C_VEL
LIN {X 0,Y 512.624,Z 298.629,A -85,B 0,C 180,E1 23733.596,E2 23733.596} C_VEL
LIN {X 0,Y 512.596,Z 298.631,A -85,B 0,C 180,E1 23730.225,E2 23730.225} C_VEL
LIN {X 0,Y 512.63,Z 298.627,A -85,B 0,C 180,E1 23726.795,E2 23726.795} C_VEL
LIN {X 0,Y 512.641,Z 298.604,A -85,B 0,C 180,E1 23723.357,E2 23723.357} C_VEL
LIN {X 0,Y 512.608,Z 298.63,A -85,B 0,C 180,E1 23719.934,E2 23719.934} C_VEL
LIN {X 0,Y 512.624,Z 298.629,A -85,B 0,C 180,E1 23716.487,E2 23716.487} C_VEL
LIN {X 0,Y 512.646,Z 298.61,A -85,B 0,C 180,E1 23713.048,E2 23713.048} C_VEL
LIN {X 0,Y 512.623,Z 298.609,A -85,B 0,C 180,E1 23709.607,E2 23709.607} C_VEL
LIN {X 0,Y 512.684,Z 298.875,A -85,B 0,C 180,E1 23709.264,E2 23709.264} C_VEL
LIN {X 0,Y 514.331,Z 303.21,A -85,B 0,C 180,E1 23708.782,E2 23708.782} C_VEL
LIN {X 0,Y 523.7,Z 325.924,A -85,B 0,C 180,E1 23706.56,E2 23706.56} C_VEL
LIN {X 0,Y 521.975,Z 379.355,A -85,B 0,C 180,E1 23703.218,E2 23703.218} C_VEL
LIN {X 0,Y 521.733,Z 389.76,A -85,B 0,C 180,E1 23702.599,E2 23702.599} C_VEL
LIN {X 0,Y 523.737,Z 405.858,A -85,B 0,C 180,E1 23702.223,E2 23702.223} C_VEL
LIN {X 0,Y 521.842,Z 612.619,A -85,B 0,C 180,E1 23699.181,E2 23699.181} C_VEL
LIN {X 0,Y 521.403,Z 654.512,A -85,B 0,C 180,E1 23698.542,E2 23698.542} C_VEL
LIN {X 0,Y 520.82,Z 675.959,A -85,B 0,C 180,E1 23698.013,E2 23698.013} C_VEL
LIN {X 0,Y 520.107,Z 696.653,A -85,B 0,C 180,E1 23697.289,E2 23697.289} C_VEL
LIN {X 0,Y 519.325,Z 714.871,A -85,B 0,C 180,E1 23696.458,E2 23696.458} C_VEL
LIN {X 0,Y 518.292,Z 733.832,A -85,B 0,C 180,E1 23695.357,E2 23695.357} C_VEL
LIN {X 0,Y 517.243,Z 751.976,A -85,B 0,C 180,E1 23694.071,E2 23694.071} C_VEL
LIN {X 0,Y 516.192,Z 769.069,A -85,B 0,C 180,E1 23692.622,E2 23692.622} C_VEL
LIN {X 0,Y 515.192,Z 785.082,A -85,B 0,C 180,E1 23691.013,E2 23691.013} C_VEL
LIN {X 0,Y 514.317,Z 799.521,A -85,B 0,C 180,E1 23689.298,E2 23689.298} C_VEL
LIN {X 0,Y 513.57,Z 812.811,A -85,B 0,C 180,E1 23687.446,E2 23687.446} C_VEL
LIN {X 0,Y 512.95,Z 825.379,A -85,B 0,C 180,E1 23685.372,E2 23685.372} C_VEL
LIN {X 0,Y 512.491,Z 836.334,A -85,B 0,C 180,E1 23683.195,E2 23683.195} C_VEL
LIN {X 0,Y 512.2,Z 845.252,A -85,B 0,C 180,E1 23681.029,E2 23681.029} C_VEL
LIN {X 0,Y 512.043,Z 852.402,A -85,B 0,C 180,E1 23678.865,E2 23678.865} C_VEL
LIN {X 0,Y 511.95,Z 858.005,A -85,B 0,C 180,E1 23676.617,E2 23676.617} C_VEL
LIN {X 0,Y 511.911,Z 861.928,A -85,B 0,C 180,E1 23674.369,E2 23674.369} C_VEL
LIN {X 0,Y 511.91,Z 864.305,A -85,B 0,C 180,E1 23672.015,E2 23672.015} C_VEL
LIN {X 0,Y 511.906,Z 864.962,A -85,B 0,C 180,E1 23669.776,E2 23669.776} C_VEL
LIN {X 0,Y 511.902,Z 864.032,A -85,B 0,C 180,E1 23667.537,E2 23667.537} C_VEL
LIN {X 0,Y 511.918,Z 861.448,A -85,B 0,C 180,E1 23665.295,E2 23665.295} C_VEL
LIN {X 0,Y 511.966,Z 857.245,A -85,B 0,C 180,E1 23663.045,E2 23663.045} C_VEL
LIN {X 0,Y 512.061,Z 851.327,A -85,B 0,C 180,E1 23660.787,E2 23660.787} C_VEL
LIN {X 0,Y 512.243,Z 844.012,A -85,B 0,C 180,E1 23658.63,E2 23658.63} C_VEL
LIN {X 0,Y 512.563,Z 834.785,A -85,B 0,C 180,E1 23656.463,E2 23656.463} C_VEL
LIN {X 0,Y 513.011,Z 824.109,A -85,B 0,C 180,E1 23654.398,E2 23654.398} C_VEL
LIN {X 0,Y 513.614,Z 812.042,A -85,B 0,C 180,E1 23652.438,E2 23652.438} C_VEL
LIN {X 0,Y 514.423,Z 797.669,A -85,B 0,C 180,E1 23650.47,E2 23650.47} C_VEL
LIN {X 0,Y 515.331,Z 782.612,A -85,B 0,C 180,E1 23648.727,E2 23648.727} C_VEL
LIN {X 0,Y 516.314,Z 767.011,A -85,B 0,C 180,E1 23647.189,E2 23647.189} C_VEL
LIN {X 0,Y 517.394,Z 749.769,A -85,B 0,C 180,E1 23645.755,E2 23645.755} C_VEL
LIN {X 0,Y 518.468,Z 731.124,A -85,B 0,C 180,E1 23644.469,E2 23644.469} C_VEL
LIN {X 0,Y 519.38,Z 713.518,A -85,B 0,C 180,E1 23643.474,E2 23643.474} C_VEL
LIN {X 0,Y 520.185,Z 694.39,A -85,B 0,C 180,E1 23642.625,E2 23642.625} C_VEL
LIN {X 0,Y 520.857,Z 674.152,A -85,B 0,C 180,E1 23641.935,E2 23641.935} C_VEL
LIN {X 0,Y 521.45,Z 652.683,A -85,B 0,C 180,E1 23641.42,E2 23641.42} C_VEL
LIN {X 0,Y 523.652,Z 413.389,A -85,B 0,C 180,E1 23637.89,E2 23637.89} C_VEL
LIN {X 0,Y 523.514,Z 402.54,A -85,B 0,C 180,E1 23637.711,E2 23637.711} C_VEL
LIN {X 0,Y 521.655,Z 388.415,A -85,B 0,C 180,E1 23637.348,E2 23637.348} C_VEL
LIN {X 0,Y 523.427,Z 334.157,A -85,B 0,C 180,E1 23633.961,E2 23633.961} C_VEL
LIN {X 0,Y 523.701,Z 325.929,A -85,B 0,C 180,E1 23633.44,E2 23633.44} C_VEL
LIN {X 0,Y 513.893,Z 302.019,A -85,B 0,C 180,E1 23631.101,E2 23631.101} C_VEL
LIN {X 0,Y 512.687,Z 298.891,A -85,B 0,C 180,E1 23630.736,E2 23630.736} C_VEL
LIN {X 0,Y 512.646,Z 298.619,A -85,B 0,C 180,E1 23629.008,E2 23629.008} C_VEL
LIN {X 0,Y 512.624,Z 298.616,A -85,B 0,C 180,E1 23625.551,E2 23625.551} C_VEL
LIN {X 0,Y 512.609,Z 298.606,A -85,B 0,C 180,E1 23622.143,E2 23622.143} C_VEL
LIN {X 0,Y 512.649,Z 298.631,A -85,B 0,C 180,E1 23618.728,E2 23618.728} C_VEL
LIN {X 0,Y 512.626,Z 298.607,A -85,B 0,C 180,E1 23615.263,E2 23615.263} C_VEL
LIN {X 0,Y 512.601,Z 298.628,A -85,B 0,C 180,E1 23611.911,E2 23611.911} C_VEL
LIN {X 0,Y 512.643,Z 298.629,A -85,B 0,C 180,E1 23608.545,E2 23608.545} C_VEL
LIN {X 0,Y 512.62,Z 298.629,A -85,B 0,C 180,E1 23605.163,E2 23605.163} C_VEL
LIN {X 0,Y 512.589,Z 298.63,A -85,B 0,C 180,E1 23601.753,E2 23601.753} C_VEL
LIN {X 0,Y 512.629,Z 298.623,A -85,B 0,C 180,E1 23598.419,E2 23598.419} C_VEL
LIN {X 0,Y 512.612,Z 298.63,A -85,B 0,C 180,E1 23595.035,E2 23595.035} C_VEL
LIN {X 0,Y 512.579,Z 298.631,A -85,B 0,C 180,E1 23591.704,E2 23591.704} C_VEL
LIN {X 0,Y 512.63,Z 298.621,A -85,B 0,C 180,E1 23588.411,E2 23588.411} C_VEL
LIN {X 0,Y 512.584,Z 298.632,A -85,B 0,C 180,E1 23585.148,E2 23585.148} C_VEL
LIN {X 0,Y 512.571,Z 298.629,A -85,B 0,C 180,E1 23581.676,E2 23581.676} C_VEL
LIN {X 0,Y 512.63,Z 298.625,A -85,B 0,C 180,E1 23578.435,E2 23578.435} C_VEL
LIN {X 0,Y 512.575,Z 298.631,A -85,B 0,C 180,E1 23575.076,E2 23575.076} C_VEL
LIN {X 0,Y 512.57,Z 298.621,A -85,B 0,C 180,E1 23571.587,E2 23571.587} C_VEL
LIN {X 0,Y 512.633,Z 298.63,A -85,B 0,C 180,E1 23568.263,E2 23568.263} C_VEL
LIN {X 0,Y 512.585,Z 298.623,A -85,B 0,C 180,E1 23564.963,E2 23564.963} C_VEL
LIN {X 0,Y 512.583,Z 298.627,A -85,B 0,C 180,E1 23561.438,E2 23561.438} C_VEL
LIN {X 0,Y 512.642,Z 298.63,A -85,B 0,C 180,E1 23558.128,E2 23558.128} C_VEL
LIN {X 0,Y 512.605,Z 298.622,A -85,B 0,C 180,E1 23554.712,E2 23554.712} C_VEL
LIN {X 0,Y 512.592,Z 298.627,A -85,B 0,C 180,E1 23551.324,E2 23551.324} C_VEL
LIN {X 0,Y 512.644,Z 298.627,A -85,B 0,C 180,E1 23547.96,E2 23547.96} C_VEL
LIN {X 0,Y 512.615,Z 298.63,A -85,B 0,C 180,E1 23544.598,E2 23544.598} C_VEL
LIN {X 0,Y 512.601,Z 298.628,A -85,B 0,C 180,E1 23541.235,E2 23541.235} C_VEL
LIN {X 0,Y 512.646,Z 298.628,A -85,B 0,C 180,E1 23537.827,E2 23537.827} C_VEL
LIN {X 0,Y 512.628,Z 298.61,A -85,B 0,C 180,E1 23534.443,E2 23534.443} C_VEL
LIN {X 0,Y 512.646,Z 298.604,A -85,B 0,C 180,E1 23534.05,E2 23534.05} C_VEL
LIN {X 0,Y 511.659,Z 298.729,A -85,B 0,C 180,E1 23533.189,E2 23533.189} C_VEL
LIN {X 0,Y 505.222,Z 299.555,A -85,B 0,C 180,E1 23530.77,E2 23530.77} C_VEL
LIN {X 0,Y 504.708,Z 299.611,A -85,B 0,C 180,E1 23530.139,E2 23530.139} C_VEL
LIN {X 0,Y 504.679,Z 299.619,A -85,B 0,C 180,E1 23526.642,E2 23526.642} C_VEL
LIN {X 0,Y 504.68,Z 299.612,A -85,B 0,C 180,E1 23523.066,E2 23523.066} C_VEL
LIN {X 0,Y 504.739,Z 299.824,A -85,B 0,C 180,E1 23521.797,E2 23521.797} C_VEL
LIN {X 0,Y 511.429,Z 319.703,A -85,B 0,C 180,E1 23519.085,E2 23519.085} C_VEL
LIN {X 0,Y 512.416,Z 323.723,A -85,B 0,C 180,E1 23518.589,E2 23518.589} C_VEL
LIN {X 0,Y 511.881,Z 338.043,A -85,B 0,C 180,E1 23517.206,E2 23517.206} C_VEL
LIN {X 0,Y 514.747,Z 351.959,A -85,B 0,C 180,E1 23516.804,E2 23516.804} C_VEL
LIN {X 0,Y 513.374,Z 549.16,A -85,B 0,C 180,E1 23514.017,E2 23514.017} C_VEL
LIN {X 0,Y 513.036,Z 567.95,A -85,B 0,C 180,E1 23513.533,E2 23513.533} C_VEL
LIN {X 0,Y 512.418,Z 586.083,A -85,B 0,C 180,E1 23512.848,E2 23512.848} C_VEL
LIN {X 0,Y 511.621,Z 603.28,A -85,B 0,C 180,E1 23511.977,E2 23511.977} C_VEL
LIN {X 0,Y 510.653,Z 619.451,A -85,B 0,C 180,E1 23510.937,E2 23510.937} C_VEL
LIN {X 0,Y 509.554,Z 635.433,A -85,B 0,C 180,E1 23509.659,E2 23509.659} C_VEL
LIN {X 0,Y 508.444,Z 650.127,A -85,B 0,C 180,E1 23508.22,E2 23508.22} C_VEL
LIN {X 0,Y 507.44,Z 662.883,A -85,B 0,C 180,E1 23506.718,E2 23506.718} C_VEL
LIN {X 0,Y 506.479,Z 675.107,A -85,B 0,C 180,E1 23504.987,E2 23504.987} C_VEL
LIN {X 0,Y 505.703,Z 685.853,A -85,B 0,C 180,E1 23503.142,E2 23503.142} C_VEL
LIN {X 0,Y 505.073,Z 695.186,A -85,B 0,C 180,E1 23501.186,E2 23501.186} C_VEL
LIN {X 0,Y 504.638,Z 703.041,A -85,B 0,C 180,E1 23499.12,E2 23499.12} C_VEL
LIN {X 0,Y 504.367,Z 709.364,A -85,B 0,C 180,E1 23496.945,E2 23496.945} C_VEL
LIN {X 0,Y 504.201,Z 714.057,A -85,B 0,C 180,E1 23494.663,E2 23494.663} C_VEL
LIN {X 0,Y 504.128,Z 716.767,A -85,B 0,C 180,E1 23492.501,E2 23492.501} C_VEL
LIN {X 0,Y 504.109,Z 717.852,A -85,B 0,C 180,E1 23490.341,E2 23490.341} C_VEL
LIN {X 0,Y 504.121,Z 717.337,A -85,B 0,C 180,E1 23488.182,E2 23488.182} C_VEL
LIN {X 0,Y 504.169,Z 715.167,A -85,B 0,C 180,E1 23485.984,E2 23485.984} C_VEL
LIN {X 0,Y 504.285,Z 711.422,A -85,B 0,C 180,E1 23483.854,E2 23483.854} C_VEL
LIN {X 0,Y 504.501,Z 706.194,A -85,B 0,C 180,E1 23481.796,E2 23481.796} C_VEL
LIN {X 0,Y 504.835,Z 699.254,A -85,B 0,C 180,E1 23479.732,E2 23479.732} C_VEL
LIN {X 0,Y 505.345,Z 690.915,A -85,B 0,C 180,E1 23477.778,E2 23477.778} C_VEL
LIN {X 0,Y 506.073,Z 680.59,A -85,B 0,C 180,E1 23475.819,E2 23475.819} C_VEL
LIN {X 0,Y 506.911,Z 669.493,A -85,B 0,C 180,E1 23474.088,E2 23474.088} C_VEL
LIN {X 0,Y 507.906,Z 657.034,A -85,B 0,C 180,E1 23472.471,E2 23472.471} C_VEL
LIN {X 0,Y 508.98,Z 643.116,A -85,B 0,C 180,E1 23470.969,E2 23470.969} C_VEL
LIN {X 0,Y 510.069,Z 628.183,A -85,B 0,C 180,E1 23469.639,E2 23469.639} C_VEL
LIN {X 0,Y 511.099,Z 612.257,A -85,B 0,C 180,E1 23468.482,E2 23468.482} C_VEL
LIN {X 0,Y 511.97,Z 596.327,A -85,B 0,C 180,E1 23467.555,E2 23467.555} C_VEL
LIN {X 0,Y 512.653,Z 579.704,A -85,B 0,C 180,E1 23466.799,E2 23466.799} C_VEL
LIN {X 0,Y 513.163,Z 561.572,A -85,B 0,C 180,E1 23466.192,E2 23466.192} C_VEL
LIN {X 0,Y 513.421,Z 543.114,A -85,B 0,C 180,E1 23465.788,E2 23465.788} C_VEL
LIN {X 0,Y 514.59,Z 350.216,A -85,B 0,C 180,E1 23463.068,E2 23463.068} C_VEL
LIN {X 0,Y 511.822,Z 337.494,A -85,B 0,C 180,E1 23462.673,E2 23462.673} C_VEL
LIN {X 0,Y 512.316,Z 322.47,A -85,B 0,C 180,E1 23461.181,E2 23461.181} C_VEL
LIN {X 0,Y 506.25,Z 304.508,A -85,B 0,C 180,E1 23458.781,E2 23458.781} C_VEL
LIN {X 0,Y 504.735,Z 299.815,A -85,B 0,C 180,E1 23458.102,E2 23458.102} C_VEL
LIN {X 0,Y 504.692,Z 299.608,A -85,B 0,C 180,E1 23454.657,E2 23454.657} C_VEL
LIN {X 0,Y 504.674,Z 299.6,A -85,B 0,C 180,E1 23451.096,E2 23451.096} C_VEL
LIN {X 0,Y 504.699,Z 299.606,A -85,B 0,C 180,E1 23447.642,E2 23447.642} C_VEL
LIN {X 0,Y 504.71,Z 299.609,A -85,B 0,C 180,E1 23444.056,E2 23444.056} C_VEL
LIN {X 0,Y 504.673,Z 299.616,A -85,B 0,C 180,E1 23440.643,E2 23440.643} C_VEL
LIN {X 0,Y 504.672,Z 299.619,A -85,B 0,C 180,E1 23437.177,E2 23437.177} C_VEL
LIN {X 0,Y 504.706,Z 299.611,A -85,B 0,C 180,E1 23433.693,E2 23433.693} C_VEL
LIN {X 0,Y 504.687,Z 299.615,A -85,B 0,C 180,E1 23430.213,E2 23430.213} C_VEL
LIN {X 0,Y 504.657,Z 299.619,A -85,B 0,C 180,E1 23426.855,E2 23426.855} C_VEL
LIN {X 0,Y 504.693,Z 299.616,A -85,B 0,C 180,E1 23423.466,E2 23423.466} C_VEL
LIN {X 0,Y 504.676,Z 299.614,A -85,B 0,C 180,E1 23420.106,E2 23420.106} C_VEL
LIN {X 0,Y 504.645,Z 299.62,A -85,B 0,C 180,E1 23416.696,E2 23416.696} C_VEL
LIN {X 0,Y 504.673,Z 299.616,A -85,B 0,C 180,E1 23413.287,E2 23413.287} C_VEL
LIN {X 0,Y 504.671,Z 299.619,A -85,B 0,C 180,E1 23409.926,E2 23409.926} C_VEL
LIN {X 0,Y 504.633,Z 299.621,A -85,B 0,C 180,E1 23406.599,E2 23406.599} C_VEL
LIN {X 0,Y 504.66,Z 299.61,A -85,B 0,C 180,E1 23403.18,E2 23403.18} C_VEL
LIN {X 0,Y 504.653,Z 299.622,A -85,B 0,C 180,E1 23399.887,E2 23399.887} C_VEL
LIN {X 0,Y 504.627,Z 299.615,A -85,B 0,C 180,E1 23396.479,E2 23396.479} C_VEL
LIN {X 0,Y 504.664,Z 299.613,A -85,B 0,C 180,E1 23393.059,E2 23393.059} C_VEL
LIN {X 0,Y 504.67,Z 299.619,A -85,B 0,C 180,E1 23389.729,E2 23389.729} C_VEL
LIN {X 0,Y 504.64,Z 299.609,A -85,B 0,C 180,E1 23386.363,E2 23386.363} C_VEL
LIN {X 0,Y 504.674,Z 299.615,A -85,B 0,C 180,E1 23382.95,E2 23382.95} C_VEL
LIN {X 0,Y 504.688,Z 299.619,A -85,B 0,C 180,E1 23379.562,E2 23379.562} C_VEL
LIN {X 0,Y 504.653,Z 299.615,A -85,B 0,C 180,E1 23376.16,E2 23376.16} C_VEL
LIN {X 0,Y 504.678,Z 299.612,A -85,B 0,C 180,E1 23372.764,E2 23372.764} C_VEL
LIN {X 0,Y 504.71,Z 299.611,A -85,B 0,C 180,E1 23369.289,E2 23369.289} C_VEL
LIN {X 0,Y 504.666,Z 299.618,A -85,B 0,C 180,E1 23365.897,E2 23365.897} C_VEL
LIN {X 0,Y 504.671,Z 299.613,A -85,B 0,C 180,E1 23362.395,E2 23362.395} C_VEL
LIN {X 0,Y 504.712,Z 299.592,A -85,B 0,C 180,E1 23359.004,E2 23359.004} C_VEL
LIN {X 0,Y 504.695,Z 299.618,A -85,B 0,C 180,E1 23355.468,E2 23355.468} C_VEL
LIN {X 0,Y 504.675,Z 299.621,A -85,B 0,C 180,E1 23352.017,E2 23352.017} C_VEL
LIN {X 0,Y 504.713,Z 299.862,A -85,B 0,C 180,E1 23349.836,E2 23349.836} C_VEL
LIN {X 0,Y 506.757,Z 305.082,A -85,B 0,C 180,E1 23349.248,E2 23349.248} C_VEL
LIN {X 0,Y 515.441,Z 326.149,A -85,B 0,C 180,E1 23347.131,E2 23347.131} C_VEL
LIN {X 0,Y 516.629,Z 329.342,A -85,B 0,C 180,E1 23346.831,E2 23346.831} C_VEL
LIN {X 0,Y 514.659,Z 383.058,A -85,B 0,C 180,E1 23343.419,E2 23343.419} C_VEL
LIN {X 0,Y 514.541,Z 389.313,A -85,B 0,C 180,E1 23343.054,E2 23343.054} C_VEL
LIN {X 0,Y 516.716,Z 406.891,A -85,B 0,C 180,E1 23342.635,E2 23342.635} C_VEL
LIN {X 0,Y 514.458,Z 621.066,A -85,B 0,C 180,E1 23339.42,E2 23339.42} C_VEL
LIN {X 0,Y 514.029,Z 654.431,A -85,B 0,C 180,E1 23338.889,E2 23338.889} C_VEL
LIN {X 0,Y 513.381,Z 675.365,A -85,B 0,C 180,E1 23338.36,E2 23338.36} C_VEL
LIN {X 0,Y 512.611,Z 695.931,A -85,B 0,C 180,E1 23337.628,E2 23337.628} C_VEL
LIN {X 0,Y 511.7,Z 715.853,A -85,B 0,C 180,E1 23336.705,E2 23336.705} C_VEL
LIN {X 0,Y 510.725,Z 734.559,A -85,B 0,C 180,E1 23335.635,E2 23335.635} C_VEL
LIN {X 0,Y 509.751,Z 752.602,A -85,B 0,C 180,E1 23334.386,E2 23334.386} C_VEL
LIN {X 0,Y 508.755,Z 767.669,A -85,B 0,C 180,E1 23333.109,E2 23333.109} C_VEL
LIN {X 0,Y 507.611,Z 784.278,A -85,B 0,C 180,E1 23331.431,E2 23331.431} C_VEL
LIN {X 0,Y 506.655,Z 798.595,A -85,B 0,C 180,E1 23329.722,E2 23329.722} C_VEL
LIN {X 0,Y 505.818,Z 812.04,A -85,B 0,C 180,E1 23327.841,E2 23327.841} C_VEL
LIN {X 0,Y 505.145,Z 824.107,A -85,B 0,C 180,E1 23325.851,E2 23325.851} C_VEL
LIN {X 0,Y 504.646,Z 834.787,A -85,B 0,C 180,E1 23323.754,E2 23323.754} C_VEL
LIN {X 0,Y 504.289,Z 844.009,A -85,B 0,C 180,E1 23321.551,E2 23321.551} C_VEL
LIN {X 0,Y 504.084,Z 851.323,A -85,B 0,C 180,E1 23319.36,E2 23319.36} C_VEL
LIN {X 0,Y 503.974,Z 857.243,A -85,B 0,C 180,E1 23317.065,E2 23317.065} C_VEL
LIN {X 0,Y 503.917,Z 861.608,A -85,B 0,C 180,E1 23314.666,E2 23314.666} C_VEL
LIN {X 0,Y 503.902,Z 864.101,A -85,B 0,C 180,E1 23312.388,E2 23312.388} C_VEL
LIN {X 0,Y 503.912,Z 864.984,A -85,B 0,C 180,E1 23310.114,E2 23310.114} C_VEL
LIN {X 0,Y 503.908,Z 864.236,A -85,B 0,C 180,E1 23307.839,E2 23307.839} C_VEL
LIN {X 0,Y 503.912,Z 861.926,A -85,B 0,C 180,E1 23305.562,E2 23305.562} C_VEL
LIN {X 0,Y 503.959,Z 858.006,A -85,B 0,C 180,E1 23303.278,E2 23303.278} C_VEL
LIN {X 0,Y 504.058,Z 852.379,A -85,B 0,C 180,E1 23300.985,E2 23300.985} C_VEL
LIN {X 0,Y 504.255,Z 844.847,A -85,B 0,C 180,E1 23298.68,E2 23298.68} C_VEL
LIN {X 0,Y 504.593,Z 835.819,A -85,B 0,C 180,E1 23296.478,E2 23296.478} C_VEL
LIN {X 0,Y 505.077,Z 825.378,A -85,B 0,C 180,E1 23294.382,E2 23294.382} C_VEL
LIN {X 0,Y 505.772,Z 812.811,A -85,B 0,C 180,E1 23292.276,E2 23292.276} C_VEL
LIN {X 0,Y 506.598,Z 799.52,A -85,B 0,C 180,E1 23290.396,E2 23290.396} C_VEL
LIN {X 0,Y 507.575,Z 784.829,A -85,B 0,C 180,E1 23288.628,E2 23288.628} C_VEL
LIN {X 0,Y 508.694,Z 768.567,A -85,B 0,C 180,E1 23286.975,E2 23286.975} C_VEL
LIN {X 0,Y 509.702,Z 753.356,A -85,B 0,C 180,E1 23285.674,E2 23285.674} C_VEL
LIN {X 0,Y 510.675,Z 735.504,A -85,B 0,C 180,E1 23284.424,E2 23284.424} C_VEL
LIN {X 0,Y 511.651,Z 717.032,A -85,B 0,C 180,E1 23283.354,E2 23283.354} C_VEL
LIN {X 0,Y 512.581,Z 696.692,A -85,B 0,C 180,E1 23282.402,E2 23282.402} C_VEL
LIN {X 0,Y 513.374,Z 675.607,A -85,B 0,C 180,E1 23281.648,E2 23281.648} C_VEL
LIN {X 0,Y 514.012,Z 654.92,A -85,B 0,C 180,E1 23281.122,E2 23281.122} C_VEL
LIN {X 0,Y 514.431,Z 623.804,A -85,B 0,C 180,E1 23280.62,E2 23280.62} C_VEL
LIN {X 0,Y 516.679,Z 409.85,A -85,B 0,C 180,E1 23277.41,E2 23277.41} C_VEL
LIN {X 0,Y 516.442,Z 403.292,A -85,B 0,C 180,E1 23277.29,E2 23277.29} C_VEL
LIN {X 0,Y 514.468,Z 387.957,A -85,B 0,C 180,E1 23276.891,E2 23276.891} C_VEL
LIN {X 0,Y 516.463,Z 333.855,A -85,B 0,C 180,E1 23273.459,E2 23273.459} C_VEL
LIN {X 0,Y 516.534,Z 328.811,A -85,B 0,C 180,E1 23273.126,E2 23273.126} C_VEL
LIN {X 0,Y 507.264,Z 306.162,A -85,B 0,C 180,E1 23270.87,E2 23270.87} C_VEL
LIN {X 0,Y 504.735,Z 299.994,A -85,B 0,C 180,E1 23270.189,E2 23270.189} C_VEL
LIN {X 0,Y 504.681,Z 299.598,A -85,B 0,C 180,E1 23269.707,E2 23269.707} C_VEL
LIN {X 0,Y 504.673,Z 299.599,A -85,B 0,C 180,E1 23266.15,E2 23266.15} C_VEL
LIN {X 0,Y 504.7,Z 299.596,A -85,B 0,C 180,E1 23262.651,E2 23262.651} C_VEL
LIN {X 0,Y 504.705,Z 299.616,A -85,B 0,C 180,E1 23259.195,E2 23259.195} C_VEL
LIN {X 0,Y 504.661,Z 299.594,A -85,B 0,C 180,E1 23255.765,E2 23255.765} C_VEL
LIN {X 0,Y 504.673,Z 299.618,A -85,B 0,C 180,E1 23252.226,E2 23252.226} C_VEL
LIN {X 0,Y 504.713,Z 299.62,A -85,B 0,C 180,E1 23248.776,E2 23248.776} C_VEL
LIN {X 0,Y 504.668,Z 299.619,A -85,B 0,C 180,E1 23245.337,E2 23245.337} C_VEL
LIN {X 0,Y 504.653,Z 299.62,A -85,B 0,C 180,E1 23241.868,E2 23241.868} C_VEL
LIN {X 0,Y 504.695,Z 299.611,A -85,B 0,C 180,E1 23238.48,E2 23238.48} C_VEL
LIN {X 0,Y 504.673,Z 299.619,A -85,B 0,C 180,E1 23235.042,E2 23235.042} C_VEL
LIN {X 0,Y 504.64,Z 299.62,A -85,B 0,C 180,E1 23231.659,E2 23231.659} C_VEL
LIN {X 0,Y 504.679,Z 299.61,A -85,B 0,C 180,E1 23228.315,E2 23228.315} C_VEL
LIN {X 0,Y 504.656,Z 299.621,A -85,B 0,C 180,E1 23225.001,E2 23225.001} C_VEL
LIN {X 0,Y 504.63,Z 299.618,A -85,B 0,C 180,E1 23221.589,E2 23221.589} C_VEL
LIN {X 0,Y 504.678,Z 299.613,A -85,B 0,C 180,E1 23218.297,E2 23218.297} C_VEL
LIN {X 0,Y 504.65,Z 299.62,A -85,B 0,C 180,E1 23214.885,E2 23214.885} C_VEL
LIN {X 0,Y 504.629,Z 299.609,A -85,B 0,C 180,E1 23211.454,E2 23211.454} C_VEL
LIN {X 0,Y 504.676,Z 299.619,A -85,B 0,C 180,E1 23208.109,E2 23208.109} C_VEL
LIN {X 0,Y 504.66,Z 299.612,A -85,B 0,C 180,E1 23204.762,E2 23204.762} C_VEL
LIN {X 0,Y 504.643,Z 299.616,A -85,B 0,C 180,E1 23201.398,E2 23201.398} C_VEL
LIN {X 0,Y 504.689,Z 299.618,A -85,B 0,C 180,E1 23197.994,E2 23197.994} C_VEL
LIN {X 0,Y 504.675,Z 299.61,A -85,B 0,C 180,E1 23194.608,E2 23194.608} C_VEL
LIN {X 0,Y 504.652,Z 299.616,A -85,B 0,C 180,E1 23191.219,E2 23191.219} C_VEL
LIN {X 0,Y 504.702,Z 299.616,A -85,B 0,C 180,E1 23187.931,E2 23187.931} C_VEL
LIN {X 0,Y 504.684,Z 299.619,A -85,B 0,C 180,E1 23184.512,E2 23184.512} C_VEL
LIN {X 0,Y 504.66,Z 299.618,A -85,B 0,C 180,E1 23181.093,E2 23181.093} C_VEL
LIN {X 0,Y 504.693,Z 299.617,A -85,B 0,C 180,E1 23177.641,E2 23177.641} C_VEL
LIN {X 0,Y 504.704,Z 299.592,A -85,B 0,C 180,E1 23174.18,E2 23174.18} C_VEL
LIN {X 0,Y 504.676,Z 299.623,A -85,B 0,C 180,E1 23170.677,E2 23170.677} C_VEL
LIN {X 0,Y 504.708,Z 299.611,A -85,B 0,C 180,E1 23170.139,E2 23170.139} C_VEL
LIN {X 0,Y 503.738,Z 299.726,A -85,B 0,C 180,E1 23169.265,E2 23169.265} C_VEL
LIN {X 0,Y 497.288,Z 300.549,A -85,B 0,C 180,E1 23166.807,E2 23166.807} C_VEL
LIN {X 0,Y 496.766,Z 300.607,A -85,B 0,C 180,E1 23166.166,E2 23166.166} C_VEL
LIN {X 0,Y 496.742,Z 300.61,A -85,B 0,C 180,E1 23162.644,E2 23162.644} C_VEL
LIN {X 0,Y 496.803,Z 300.914,A -85,B 0,C 180,E1 23162.336,E2 23162.336} C_VEL
LIN {X 0,Y 503.421,Z 320.289,A -85,B 0,C 180,E1 23159.639,E2 23159.639} C_VEL
LIN {X 0,Y 505.217,Z 326.167,A -85,B 0,C 180,E1 23158.874,E2 23158.874} C_VEL
LIN {X 0,Y 504.756,Z 338.534,A -85,B 0,C 180,E1 23157.677,E2 23157.677} C_VEL
LIN {X 0,Y 507.823,Z 353.46,A -85,B 0,C 180,E1 23157.237,E2 23157.237} C_VEL
LIN {X 0,Y 506.34,Z 550.11,A -85,B 0,C 180,E1 23154.433,E2 23154.433} C_VEL
LIN {X 0,Y 505.988,Z 568.991,A -85,B 0,C 180,E1 23153.943,E2 23153.943} C_VEL
LIN {X 0,Y 505.342,Z 587.22,A -85,B 0,C 180,E1 23153.248,E2 23153.248} C_VEL
LIN {X 0,Y 504.503,Z 604.507,A -85,B 0,C 180,E1 23152.365,E2 23152.365} C_VEL
LIN {X 0,Y 503.482,Z 620.785,A -85,B 0,C 180,E1 23151.31,E2 23151.31} C_VEL
LIN {X 0,Y 502.336,Z 636.582,A -85,B 0,C 180,E1 23150.035,E2 23150.035} C_VEL
LIN {X 0,Y 501.163,Z 650.98,A -85,B 0,C 180,E1 23148.615,E2 23148.615} C_VEL
LIN {X 0,Y 500.057,Z 663.784,A -85,B 0,C 180,E1 23147.093,E2 23147.093} C_VEL
LIN {X 0,Y 498.982,Z 676.037,A -85,B 0,C 180,E1 23145.337,E2 23145.337} C_VEL
LIN {X 0,Y 498.102,Z 686.807,A -85,B 0,C 180,E1 23143.465,E2 23143.465} C_VEL
LIN {X 0,Y 497.375,Z 696.144,A -85,B 0,C 180,E1 23141.479,E2 23141.479} C_VEL
LIN {X 0,Y 496.862,Z 704.015,A -85,B 0,C 180,E1 23139.381,E2 23139.381} C_VEL
LIN {X 0,Y 496.546,Z 710.089,A -85,B 0,C 180,E1 23137.288,E2 23137.288} C_VEL
LIN {X 0,Y 496.333,Z 714.727,A -85,B 0,C 180,E1 23135.085,E2 23135.085} C_VEL
LIN {X 0,Y 496.233,Z 717.667,A -85,B 0,C 180,E1 23132.887,E2 23132.887} C_VEL
LIN {X 0,Y 496.205,Z 718.991,A -85,B 0,C 180,E1 23130.693,E2 23130.693} C_VEL
LIN {X 0,Y 496.209,Z 718.732,A -85,B 0,C 180,E1 23128.499,E2 23128.499} C_VEL
LIN {X 0,Y 496.259,Z 716.885,A -85,B 0,C 180,E1 23126.304,E2 23126.304} C_VEL
LIN {X 0,Y 496.39,Z 713.394,A -85,B 0,C 180,E1 23124.104,E2 23124.104} C_VEL
LIN {X 0,Y 496.644,Z 708.164,A -85,B 0,C 180,E1 23121.899,E2 23121.899} C_VEL
LIN {X 0,Y 497.035,Z 701.064,A -85,B 0,C 180,E1 23119.687,E2 23119.687} C_VEL
LIN {X 0,Y 497.603,Z 692.919,A -85,B 0,C 180,E1 23117.703,E2 23117.703} C_VEL
LIN {X 0,Y 498.407,Z 682.823,A -85,B 0,C 180,E1 23115.715,E2 23115.715} C_VEL
LIN {X 0,Y 499.319,Z 671.974,A -85,B 0,C 180,E1 23113.959,E2 23113.959} C_VEL
LIN {X 0,Y 500.393,Z 659.804,A -85,B 0,C 180,E1 23112.32,E2 23112.32} C_VEL
LIN {X 0,Y 501.545,Z 646.213,A -85,B 0,C 180,E1 23110.796,E2 23110.796} C_VEL
LIN {X 0,Y 502.752,Z 630.927,A -85,B 0,C 180,E1 23109.39,E2 23109.39} C_VEL
LIN {X 0,Y 503.84,Z 615.244,A -85,B 0,C 180,E1 23108.217,E2 23108.217} C_VEL
LIN {X 0,Y 504.815,Z 598.584,A -85,B 0,C 180,E1 23107.219,E2 23107.219} C_VEL
LIN {X 0,Y 505.561,Z 581.515,A -85,B 0,C 180,E1 23106.423,E2 23106.423} C_VEL
LIN {X 0,Y 506.118,Z 562.925,A -85,B 0,C 180,E1 23105.789,E2 23105.789} C_VEL
LIN {X 0,Y 506.384,Z 544.23,A -85,B 0,C 180,E1 23105.374,E2 23105.374} C_VEL
LIN {X 0,Y 507.687,Z 351.726,A -85,B 0,C 180,E1 23102.635,E2 23102.635} C_VEL
LIN {X 0,Y 504.693,Z 337.826,A -85,B 0,C 180,E1 23102.19,E2 23102.19} C_VEL
LIN {X 0,Y 505.226,Z 325.83,A -85,B 0,C 180,E1 23100.997,E2 23100.997} C_VEL
LIN {X 0,Y 498.839,Z 306.698,A -85,B 0,C 180,E1 23098.415,E2 23098.415} C_VEL
LIN {X 0,Y 496.779,Z 300.776,A -85,B 0,C 180,E1 23097.529,E2 23097.529} C_VEL
LIN {X 0,Y 496.768,Z 300.601,A -85,B 0,C 180,E1 23094.149,E2 23094.149} C_VEL
LIN {X 0,Y 496.748,Z 300.59,A -85,B 0,C 180,E1 23090.617,E2 23090.617} C_VEL
LIN {X 0,Y 496.735,Z 300.589,A -85,B 0,C 180,E1 23087.112,E2 23087.112} C_VEL
LIN {X 0,Y 496.76,Z 300.607,A -85,B 0,C 180,E1 23083.567,E2 23083.567} C_VEL
LIN {X 0,Y 496.771,Z 300.603,A -85,B 0,C 180,E1 23080.096,E2 23080.096} C_VEL
LIN {X 0,Y 496.728,Z 300.606,A -85,B 0,C 180,E1 23076.715,E2 23076.715} C_VEL
LIN {X 0,Y 496.728,Z 300.608,A -85,B 0,C 180,E1 23073.14,E2 23073.14} C_VEL
LIN {X 0,Y 496.772,Z 300.598,A -85,B 0,C 180,E1 23069.678,E2 23069.678} C_VEL
LIN {X 0,Y 496.744,Z 300.606,A -85,B 0,C 180,E1 23066.156,E2 23066.156} C_VEL
LIN {X 0,Y 496.712,Z 300.609,A -85,B 0,C 180,E1 23062.736,E2 23062.736} C_VEL
LIN {X 0,Y 496.73,Z 300.601,A -85,B 0,C 180,E1 23059.263,E2 23059.263} C_VEL
LIN {X 0,Y 496.756,Z 300.607,A -85,B 0,C 180,E1 23055.829,E2 23055.829} C_VEL
LIN {X 0,Y 496.702,Z 300.607,A -85,B 0,C 180,E1 23052.439,E2 23052.439} C_VEL
LIN {X 0,Y 496.704,Z 300.597,A -85,B 0,C 180,E1 23048.917,E2 23048.917} C_VEL
LIN {X 0,Y 496.757,Z 300.61,A -85,B 0,C 180,E1 23045.544,E2 23045.544} C_VEL
LIN {X 0,Y 496.703,Z 300.6,A -85,B 0,C 180,E1 23042.077,E2 23042.077} C_VEL
LIN {X 0,Y 496.688,Z 300.606,A -85,B 0,C 180,E1 23038.616,E2 23038.616} C_VEL
LIN {X 0,Y 496.73,Z 300.61,A -85,B 0,C 180,E1 23035.151,E2 23035.151} C_VEL
LIN {X 0,Y 496.724,Z 300.6,A -85,B 0,C 180,E1 23031.784,E2 23031.784} C_VEL
LIN {X 0,Y 496.7,Z 300.61,A -85,B 0,C 180,E1 23028.387,E2 23028.387} C_VEL
LIN {X 0,Y 496.731,Z 300.609,A -85,B 0,C 180,E1 23024.95,E2 23024.95} C_VEL
LIN {X 0,Y 496.746,Z 300.6,A -85,B 0,C 180,E1 23021.578,E2 23021.578} C_VEL
LIN {X 0,Y 496.714,Z 300.608,A -85,B 0,C 180,E1 23018.116,E2 23018.116} C_VEL
LIN {X 0,Y 496.725,Z 300.608,A -85,B 0,C 180,E1 23014.612,E2 23014.612} C_VEL
LIN {X 0,Y 496.772,Z 300.607,A -85,B 0,C 180,E1 23011.115,E2 23011.115} C_VEL
LIN {X 0,Y 496.742,Z 300.608,A -85,B 0,C 180,E1 23007.628,E2 23007.628} C_VEL
LIN {X 0,Y 496.721,Z 300.58,A -85,B 0,C 180,E1 23004.144,E2 23004.144} C_VEL
LIN {X 0,Y 496.753,Z 300.605,A -85,B 0,C 180,E1 23000.652,E2 23000.652} C_VEL
LIN {X 0,Y 496.77,Z 300.588,A -85,B 0,C 180,E1 22997.105,E2 22997.105} C_VEL
LIN {X 0,Y 496.747,Z 300.584,A -85,B 0,C 180,E1 22993.564,E2 22993.564} C_VEL
LIN {X 0,Y 496.783,Z 300.823,A -85,B 0,C 180,E1 22990.433,E2 22990.433} C_VEL
LIN {X 0,Y 498.108,Z 304.176,A -85,B 0,C 180,E1 22990.023,E2 22990.023} C_VEL
LIN {X 0,Y 507.808,Z 327.665,A -85,B 0,C 180,E1 22987.589,E2 22987.589} C_VEL
LIN {X 0,Y 509.568,Z 332.753,A -85,B 0,C 180,E1 22987.11,E2 22987.11} C_VEL
LIN {X 0,Y 507.393,Z 385.651,A -85,B 0,C 180,E1 22983.697,E2 22983.697} C_VEL
LIN {X 0,Y 507.432,Z 389.258,A -85,B 0,C 180,E1 22983.512,E2 22983.512} C_VEL
LIN {X 0,Y 509.721,Z 408.002,A -85,B 0,C 180,E1 22983.057,E2 22983.057} C_VEL
LIN {X 0,Y 507.125,Z 625.41,A -85,B 0,C 180,E1 22979.728,E2 22979.728} C_VEL
LIN {X 0,Y 506.653,Z 654.921,A -85,B 0,C 180,E1 22979.232,E2 22979.232} C_VEL
LIN {X 0,Y 505.933,Z 675.538,A -85,B 0,C 180,E1 22978.691,E2 22978.691} C_VEL
LIN {X 0,Y 505.099,Z 695.941,A -85,B 0,C 180,E1 22977.946,E2 22977.946} C_VEL
LIN {X 0,Y 504.034,Z 717.336,A -85,B 0,C 180,E1 22976.924,E2 22976.924} C_VEL
LIN {X 0,Y 502.863,Z 737.943,A -85,B 0,C 180,E1 22975.686,E2 22975.686} C_VEL
LIN {X 0,Y 501.734,Z 756.879,A -85,B 0,C 180,E1 22974.296,E2 22974.296} C_VEL
LIN {X 0,Y 500.647,Z 774.041,A -85,B 0,C 180,E1 22972.795,E2 22972.795} C_VEL
LIN {X 0,Y 499.69,Z 788.423,A -85,B 0,C 180,E1 22971.295,E2 22971.295} C_VEL
LIN {X 0,Y 498.704,Z 802.24,A -85,B 0,C 180,E1 22969.558,E2 22969.558} C_VEL
LIN {X 0,Y 497.792,Z 815.873,A -85,B 0,C 180,E1 22967.534,E2 22967.534} C_VEL
LIN {X 0,Y 497.08,Z 827.917,A -85,B 0,C 180,E1 22965.397,E2 22965.397} C_VEL
LIN {X 0,Y 496.574,Z 837.876,A -85,B 0,C 180,E1 22963.27,E2 22963.27} C_VEL
LIN {X 0,Y 496.237,Z 846.465,A -85,B 0,C 180,E1 22961.035,E2 22961.035} C_VEL
LIN {X 0,Y 496.043,Z 853.594,A -85,B 0,C 180,E1 22958.695,E2 22958.695} C_VEL
LIN {X 0,Y 495.949,Z 858.727,A -85,B 0,C 180,E1 22956.482,E2 22956.482} C_VEL
LIN {X 0,Y 495.915,Z 862.405,A -85,B 0,C 180,E1 22954.162,E2 22954.162} C_VEL
LIN {X 0,Y 495.908,Z 864.44,A -85,B 0,C 180,E1 22951.849,E2 22951.849} C_VEL
LIN {X 0,Y 495.901,Z 864.894,A -85,B 0,C 180,E1 22949.422,E2 22949.422} C_VEL
LIN {X 0,Y 495.915,Z 863.732,A -85,B 0,C 180,E1 22947.111,E2 22947.111} C_VEL
LIN {X 0,Y 495.931,Z 860.968,A -85,B 0,C 180,E1 22944.795,E2 22944.795} C_VEL
LIN {X 0,Y 495.989,Z 856.482,A -85,B 0,C 180,E1 22942.471,E2 22942.471} C_VEL
LIN {X 0,Y 496.124,Z 850.267,A -85,B 0,C 180,E1 22940.137,E2 22940.137} C_VEL
LIN {X 0,Y 496.391,Z 842.176,A -85,B 0,C 180,E1 22937.79,E2 22937.79} C_VEL
LIN {X 0,Y 496.806,Z 833.135,A -85,B 0,C 180,E1 22935.668,E2 22935.668} C_VEL
LIN {X 0,Y 497.423,Z 821.957,A -85,B 0,C 180,E1 22933.497,E2 22933.497} C_VEL
LIN {X 0,Y 498.244,Z 808.955,A -85,B 0,C 180,E1 22931.394,E2 22931.394} C_VEL
LIN {X 0,Y 499.224,Z 794.89,A -85,B 0,C 180,E1 22929.483,E2 22929.483} C_VEL
LIN {X 0,Y 500.184,Z 781.316,A -85,B 0,C 180,E1 22927.926,E2 22927.926} C_VEL
LIN {X 0,Y 501.2,Z 765.293,A -85,B 0,C 180,E1 22926.409,E2 22926.409} C_VEL
LIN {X 0,Y 502.312,Z 747.42,A -85,B 0,C 180,E1 22924.978,E2 22924.978} C_VEL
LIN {X 0,Y 503.421,Z 728.435,A -85,B 0,C 180,E1 22923.711,E2 22923.711} C_VEL
LIN {X 0,Y 504.487,Z 708.483,A -85,B 0,C 180,E1 22922.626,E2 22922.626} C_VEL
LIN {X 0,Y 505.373,Z 689.011,A -85,B 0,C 180,E1 22921.781,E2 22921.781} C_VEL
LIN {X 0,Y 506.229,Z 667.949,A -85,B 0,C 180,E1 22921.089,E2 22921.089} C_VEL
LIN {X 0,Y 506.843,Z 646.696,A -85,B 0,C 180,E1 22920.605,E2 22920.605} C_VEL
LIN {X 0,Y 509.576,Z 418.361,A -85,B 0,C 180,E1 22917.104,E2 22917.104} C_VEL
LIN {X 0,Y 509.53,Z 404.975,A -85,B 0,C 180,E1 22916.881,E2 22916.881} C_VEL
LIN {X 0,Y 507.314,Z 387.543,A -85,B 0,C 180,E1 22916.424,E2 22916.424} C_VEL
LIN {X 0,Y 509.493,Z 334.564,A -85,B 0,C 180,E1 22913.008,E2 22913.008} C_VEL
LIN {X 0,Y 509.381,Z 331.679,A -85,B 0,C 180,E1 22912.803,E2 22912.803} C_VEL
LIN {X 0,Y 500.614,Z 310.145,A -85,B 0,C 180,E1 22910.618,E2 22910.618} C_VEL
LIN {X 0,Y 496.816,Z 301.036,A -85,B 0,C 180,E1 22909.608,E2 22909.608} C_VEL
LIN {X 0,Y 496.77,Z 300.586,A -85,B 0,C 180,E1 22909.3,E2 22909.3} C_VEL
LIN {X 0,Y 496.735,Z 300.588,A -85,B 0,C 180,E1 22905.772,E2 22905.772} C_VEL
LIN {X 0,Y 496.733,Z 300.581,A -85,B 0,C 180,E1 22902.208,E2 22902.208} C_VEL
LIN {X 0,Y 496.772,Z 300.608,A -85,B 0,C 180,E1 22898.752,E2 22898.752} C_VEL
LIN {X 0,Y 496.754,Z 300.582,A -85,B 0,C 180,E1 22895.198,E2 22895.198} C_VEL
LIN {X 0,Y 496.722,Z 300.605,A -85,B 0,C 180,E1 22891.829,E2 22891.829} C_VEL
LIN {X 0,Y 496.746,Z 300.605,A -85,B 0,C 180,E1 22888.361,E2 22888.361} C_VEL
LIN {X 0,Y 496.771,Z 300.608,A -85,B 0,C 180,E1 22884.809,E2 22884.809} C_VEL
LIN {X 0,Y 496.721,Z 300.607,A -85,B 0,C 180,E1 22881.367,E2 22881.367} C_VEL
LIN {X 0,Y 496.71,Z 300.605,A -85,B 0,C 180,E1 22877.805,E2 22877.805} C_VEL
LIN {X 0,Y 496.754,Z 300.599,A -85,B 0,C 180,E1 22874.453,E2 22874.453} C_VEL
LIN {X 0,Y 496.727,Z 300.608,A -85,B 0,C 180,E1 22871.024,E2 22871.024} C_VEL
LIN {X 0,Y 496.697,Z 300.603,A -85,B 0,C 180,E1 22867.635,E2 22867.635} C_VEL
LIN {X 0,Y 496.735,Z 300.604,A -85,B 0,C 180,E1 22864.271,E2 22864.271} C_VEL
LIN {X 0,Y 496.727,Z 300.606,A -85,B 0,C 180,E1 22860.807,E2 22860.807} C_VEL
LIN {X 0,Y 496.686,Z 300.601,A -85,B 0,C 180,E1 22857.461,E2 22857.461} C_VEL
LIN {X 0,Y 496.715,Z 300.61,A -85,B 0,C 180,E1 22853.991,E2 22853.991} C_VEL
LIN {X 0,Y 496.723,Z 300.597,A -85,B 0,C 180,E1 22850.733,E2 22850.733} C_VEL
LIN {X 0,Y 496.695,Z 300.609,A -85,B 0,C 180,E1 22847.325,E2 22847.325} C_VEL
LIN {X 0,Y 496.725,Z 300.609,A -85,B 0,C 180,E1 22843.872,E2 22843.872} C_VEL
LIN {X 0,Y 496.759,Z 300.597,A -85,B 0,C 180,E1 22840.381,E2 22840.381} C_VEL
LIN {X 0,Y 496.712,Z 300.61,A -85,B 0,C 180,E1 22837.013,E2 22837.013} C_VEL
LIN {X 0,Y 496.718,Z 300.608,A -85,B 0,C 180,E1 22833.457,E2 22833.457} C_VEL
LIN {X 0,Y 496.775,Z 300.599,A -85,B 0,C 180,E1 22830.056,E2 22830.056} C_VEL
LIN {X 0,Y 496.745,Z 300.604,A -85,B 0,C 180,E1 22826.529,E2 22826.529} C_VEL
LIN {X 0,Y 496.723,Z 300.608,A -85,B 0,C 180,E1 22823.044,E2 22823.044} C_VEL
LIN {X 0,Y 496.742,Z 300.605,A -85,B 0,C 180,E1 22819.537,E2 22819.537} C_VEL
LIN {X 0,Y 496.771,Z 300.6,A -85,B 0,C 180,E1 22816.021,E2 22816.021} C_VEL
LIN {X 0,Y 496.742,Z 300.592,A -85,B 0,C 180,E1 22812.549,E2 22812.549} C_VEL
LIN {X 0,Y 496.731,Z 300.589,A -85,B 0,C 180,E1 22809.015,E2 22809.015} C_VEL
LIN {X 0,Y 496.766,Z 300.607,A -85,B 0,C 180,E1 22806.166,E2 22806.166} C_VEL
LIN {X 0,Y 495.775,Z 300.723,A -85,B 0,C 180,E1 22805.575,E2 22805.575} C_VEL
LIN {X 0,Y 489.373,Z 301.503,A -85,B 0,C 180,E1 22803.971,E2 22803.971} C_VEL
LIN {X 0,Y 488.825,Z 301.575,A -85,B 0,C 180,E1 22803.535,E2 22803.535} C_VEL
LIN {X 0,Y 488.844,Z 301.894,A -85,B 0,C 180,E1 22802.925,E2 22802.925} C_VEL
LIN {X 0,Y 495.742,Z 321.797,A -85,B 0,C 180,E1 22800.088,E2 22800.088} C_VEL
LIN {X 0,Y 498.02,Z 328.793,A -85,B 0,C 180,E1 22799.151,E2 22799.151} C_VEL
LIN {X 0,Y 497.67,Z 339.087,A -85,B 0,C 180,E1 22798.159,E2 22798.159} C_VEL
LIN {X 0,Y 500.93,Z 354.775,A -85,B 0,C 180,E1 22797.684,E2 22797.684} C_VEL
LIN {X 0,Y 499.307,Z 551.109,A -85,B 0,C 180,E1 22794.855,E2 22794.855} C_VEL
LIN {X 0,Y 498.934,Z 570.008,A -85,B 0,C 180,E1 22794.358,E2 22794.358} C_VEL
LIN {X 0,Y 498.261,Z 588.121,A -85,B 0,C 180,E1 22793.661,E2 22793.661} C_VEL
LIN {X 0,Y 497.371,Z 605.484,A -85,B 0,C 180,E1 22792.766,E2 22792.766} C_VEL
LIN {X 0,Y 496.289,Z 621.829,A -85,B 0,C 180,E1 22791.696,E2 22791.696} C_VEL
LIN {X 0,Y 495.057,Z 637.793,A -85,B 0,C 180,E1 22790.395,E2 22790.395} C_VEL
LIN {X 0,Y 493.846,Z 651.827,A -85,B 0,C 180,E1 22789.001,E2 22789.001} C_VEL
LIN {X 0,Y 492.585,Z 665.464,A -85,B 0,C 180,E1 22787.36,E2 22787.36} C_VEL
LIN {X 0,Y 491.425,Z 677.665,A -85,B 0,C 180,E1 22785.579,E2 22785.579} C_VEL
LIN {X 0,Y 490.457,Z 688.347,A -85,B 0,C 180,E1 22783.679,E2 22783.679} C_VEL
LIN {X 0,Y 489.651,Z 697.598,A -85,B 0,C 180,E1 22781.663,E2 22781.663} C_VEL
LIN {X 0,Y 489.071,Z 705.39,A -85,B 0,C 180,E1 22779.532,E2 22779.532} C_VEL
LIN {X 0,Y 488.685,Z 711.677,A -85,B 0,C 180,E1 22777.288,E2 22777.288} C_VEL
LIN {X 0,Y 488.438,Z 716.36,A -85,B 0,C 180,E1 22774.932,E2 22774.932} C_VEL
LIN {X 0,Y 488.324,Z 719.198,A -85,B 0,C 180,E1 22772.582,E2 22772.582} C_VEL
LIN {X 0,Y 488.291,Z 720.256,A -85,B 0,C 180,E1 22770.352,E2 22770.352} C_VEL
LIN {X 0,Y 488.309,Z 719.751,A -85,B 0,C 180,E1 22768.123,E2 22768.123} C_VEL
LIN {X 0,Y 488.383,Z 717.672,A -85,B 0,C 180,E1 22765.891,E2 22765.891} C_VEL
LIN {X 0,Y 488.554,Z 713.959,A -85,B 0,C 180,E1 22763.655,E2 22763.655} C_VEL
LIN {X 0,Y 488.876,Z 708.516,A -85,B 0,C 180,E1 22761.414,E2 22761.414} C_VEL
LIN {X 0,Y 489.338,Z 701.622,A -85,B 0,C 180,E1 22759.284,E2 22759.284} C_VEL
LIN {X 0,Y 490.019,Z 693.261,A -85,B 0,C 180,E1 22757.25,E2 22757.25} C_VEL
LIN {X 0,Y 490.925,Z 683.109,A -85,B 0,C 180,E1 22755.251,E2 22755.251} C_VEL
LIN {X 0,Y 491.955,Z 672.054,A -85,B 0,C 180,E1 22753.469,E2 22753.469} C_VEL
LIN {X 0,Y 493.138,Z 659.594,A -85,B 0,C 180,E1 22751.806,E2 22751.806} C_VEL
LIN {X 0,Y 494.334,Z 646.199,A -85,B 0,C 180,E1 22750.32,E2 22750.32} C_VEL
LIN {X 0,Y 495.572,Z 631.291,A -85,B 0,C 180,E1 22748.954,E2 22748.954} C_VEL
LIN {X 0,Y 496.73,Z 615.382,A -85,B 0,C 180,E1 22747.765,E2 22747.765} C_VEL
LIN {X 0,Y 497.703,Z 599.514,A -85,B 0,C 180,E1 22746.812,E2 22746.812} C_VEL
LIN {X 0,Y 498.495,Z 582.352,A -85,B 0,C 180,E1 22746.005,E2 22746.005} C_VEL
LIN {X 0,Y 499.076,Z 563.889,A -85,B 0,C 180,E1 22745.37,E2 22745.37} C_VEL
LIN {X 0,Y 499.352,Z 545.212,A -85,B 0,C 180,E1 22744.95,E2 22744.95} C_VEL
LIN {X 0,Y 500.791,Z 353.157,A -85,B 0,C 180,E1 22742.188,E2 22742.188} C_VEL
LIN {X 0,Y 497.596,Z 338.367,A -85,B 0,C 180,E1 22741.709,E2 22741.709} C_VEL
LIN {X 0,Y 497.97,Z 328.618,A -85,B 0,C 180,E1 22740.732,E2 22740.732} C_VEL
LIN {X 0,Y 491.564,Z 309.601,A -85,B 0,C 180,E1 22738.115,E2 22738.115} C_VEL
LIN {X 0,Y 488.836,Z 301.801,A -85,B 0,C 180,E1 22736.953,E2 22736.953} C_VEL
LIN {X 0,Y 488.821,Z 301.599,A -85,B 0,C 180,E1 22733.618,E2 22733.618} C_VEL
LIN {X 0,Y 488.832,Z 301.582,A -85,B 0,C 180,E1 22730.041,E2 22730.041} C_VEL
LIN {X 0,Y 488.806,Z 301.568,A -85,B 0,C 180,E1 22726.566,E2 22726.566} C_VEL
LIN {X 0,Y 488.795,Z 301.598,A -85,B 0,C 180,E1 22723.093,E2 22723.093} C_VEL
LIN {X 0,Y 488.83,Z 301.598,A -85,B 0,C 180,E1 22719.656,E2 22719.656} C_VEL
LIN {X 0,Y 488.827,Z 301.593,A -85,B 0,C 180,E1 22716.092,E2 22716.092} C_VEL
LIN {X 0,Y 488.788,Z 301.595,A -85,B 0,C 180,E1 22712.568,E2 22712.568} C_VEL
LIN {X 0,Y 488.784,Z 301.593,A -85,B 0,C 180,E1 22709,E2 22709} C_VEL
LIN {X 0,Y 488.822,Z 301.587,A -85,B 0,C 180,E1 22705.569,E2 22705.569} C_VEL
LIN {X 0,Y 488.805,Z 301.596,A -85,B 0,C 180,E1 22702.09,E2 22702.09} C_VEL
LIN {X 0,Y 488.769,Z 301.592,A -85,B 0,C 180,E1 22698.61,E2 22698.61} C_VEL
LIN {X 0,Y 488.776,Z 301.588,A -85,B 0,C 180,E1 22695.058,E2 22695.058} C_VEL
LIN {X 0,Y 488.818,Z 301.596,A -85,B 0,C 180,E1 22691.684,E2 22691.684} C_VEL
LIN {X 0,Y 488.765,Z 301.585,A -85,B 0,C 180,E1 22688.233,E2 22688.233} C_VEL
LIN {X 0,Y 488.755,Z 301.597,A -85,B 0,C 180,E1 22684.694,E2 22684.694} C_VEL
LIN {X 0,Y 488.797,Z 301.596,A -85,B 0,C 180,E1 22681.29,E2 22681.29} C_VEL
LIN {X 0,Y 488.775,Z 301.592,A -85,B 0,C 180,E1 22677.89,E2 22677.89} C_VEL
LIN {X 0,Y 488.754,Z 301.599,A -85,B 0,C 180,E1 22674.483,E2 22674.483} C_VEL
LIN {X 0,Y 488.789,Z 301.592,A -85,B 0,C 180,E1 22671.057,E2 22671.057} C_VEL
LIN {X 0,Y 488.805,Z 301.592,A -85,B 0,C 180,E1 22667.598,E2 22667.598} C_VEL
LIN {X 0,Y 488.767,Z 301.599,A -85,B 0,C 180,E1 22664.212,E2 22664.212} C_VEL
